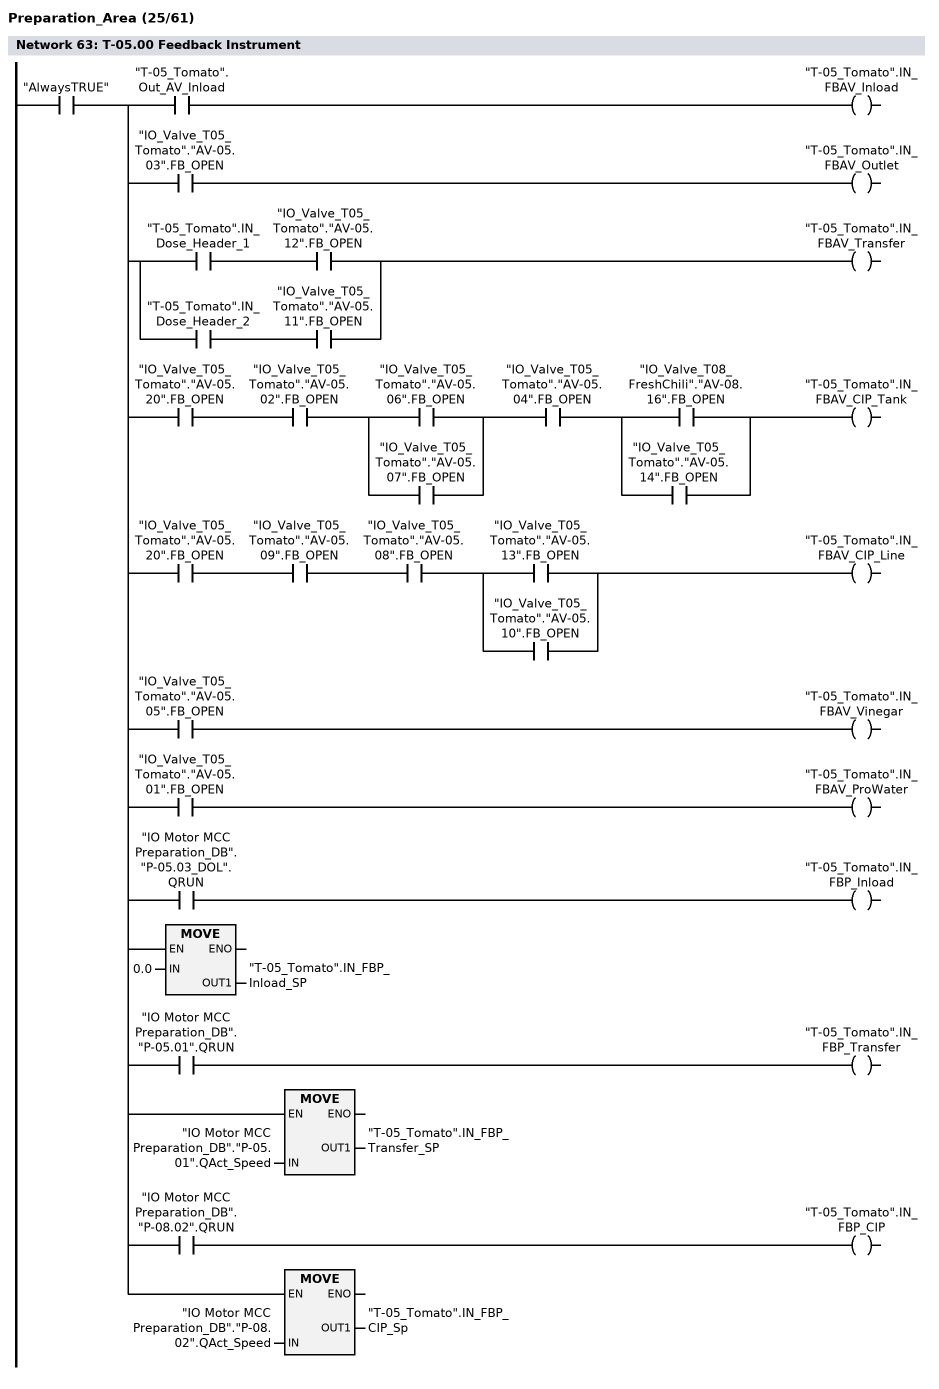
   RUNG wire#powerrail
      Contact( "AlwaysTRUE" )
      wire#w1
      Contact( "T-05_Tomato".Out_AV_Inload )
      Coil( "T-05_Tomato".IN_FBAV_Inload )
   END_RUNG
   RUNG wire#w1
      Contact( "IO_Valve_T05_Tomato"."AV-05.03".FB_OPEN )
      Coil( "T-05_Tomato".IN_FBAV_Outlet )
   END_RUNG
   RUNG wire#w1
      Contact( "T-05_Tomato".IN_Dose_Header_1 )
      Contact( "IO_Valve_T05_Tomato"."AV-05.12".FB_OPEN )
      wire#w2
      Coil( "T-05_Tomato".IN_FBAV_Transfer )
   END_RUNG
   RUNG wire#w1
      Contact( "T-05_Tomato".IN_Dose_Header_2 )
      Contact( "IO_Valve_T05_Tomato"."AV-05.11".FB_OPEN )
   END_RUNG wire#w2
   RUNG wire#w1
      Contact( "IO_Valve_T05_Tomato"."AV-05.20".FB_OPEN )
      Contact( "IO_Valve_T05_Tomato"."AV-05.02".FB_OPEN )
      wire#w3
      Contact( "IO_Valve_T05_Tomato"."AV-05.06".FB_OPEN )
      wire#w4
      Contact( "IO_Valve_T05_Tomato"."AV-05.04".FB_OPEN )
      wire#w5
      Contact( "IO_Valve_T08_FreshChili"."AV-08.16".FB_OPEN )
      wire#w6
      Coil( "T-05_Tomato".IN_FBAV_CIP_Tank )
   END_RUNG
   RUNG wire#w3
      Contact( "IO_Valve_T05_Tomato"."AV-05.07".FB_OPEN )
   END_RUNG wire#w4
   RUNG wire#w5
      Contact( "IO_Valve_T05_Tomato"."AV-05.14".FB_OPEN )
   END_RUNG wire#w6
   RUNG wire#w1
      Contact( "IO_Valve_T05_Tomato"."AV-05.20".FB_OPEN )
      Contact( "IO_Valve_T05_Tomato"."AV-05.09".FB_OPEN )
      Contact( "IO_Valve_T05_Tomato"."AV-05.08".FB_OPEN )
      wire#w7
      Contact( "IO_Valve_T05_Tomato"."AV-05.13".FB_OPEN )
      wire#w8
      Coil( "T-05_Tomato".IN_FBAV_CIP_Line )
   END_RUNG
   RUNG wire#w7
      Contact( "IO_Valve_T05_Tomato"."AV-05.10".FB_OPEN )
   END_RUNG wire#w8
   RUNG wire#w1
      Contact( "IO_Valve_T05_Tomato"."AV-05.05".FB_OPEN )
      Coil( "T-05_Tomato".IN_FBAV_Vinegar )
   END_RUNG
   RUNG wire#w1
      Contact( "IO_Valve_T05_Tomato"."AV-05.01".FB_OPEN )
      Coil( "T-05_Tomato".IN_FBAV_ProWater )
   END_RUNG
   RUNG wire#w1
      Contact( "IO Motor MCC Preparation_DB"."P-05.03_DOL".QRUN )
      Coil( "T-05_Tomato".IN_FBP_Inload )
   END_RUNG
   RUNG wire#w1
      Move(in := 0.0, out1 => "T-05_Tomato".IN_FBP_Inload_SP)
   END_RUNG
   RUNG wire#w1
      Contact( "IO Motor MCC Preparation_DB"."P-05.01".QRUN )
      Coil( "T-05_Tomato".IN_FBP_Transfer )
   END_RUNG
   RUNG wire#w1
      Move(in := "IO Motor MCC Preparation_DB"."P-05.01".QAct_Speed, out1 => "T-05_Tomato".IN_FBP_Transfer_SP)
   END_RUNG
   RUNG wire#w1
      Contact( "IO Motor MCC Preparation_DB"."P-08.02".QRUN )
      Coil( "T-05_Tomato".IN_FBP_CIP )
   END_RUNG
   RUNG wire#w1
      Move(in := "IO Motor MCC Preparation_DB"."P-08.02".QAct_Speed, out1 => "T-05_Tomato".IN_FBP_CIP_Sp)
   END_RUNG
   // the same network as SCL:
   "T-05_Tomato".IN_FBAV_Inload := "AlwaysTRUE" AND "T-05_Tomato".Out_AV_Inload;
   "T-05_Tomato".IN_FBAV_Outlet := "AlwaysTRUE" AND "IO_Valve_T05_Tomato"."AV-05.03".FB_OPEN;
   "T-05_Tomato".IN_FBAV_Transfer := "AlwaysTRUE" AND (("T-05_Tomato".IN_Dose_Header_1 AND "IO_Valve_T05_Tomato"."AV-05.12".FB_OPEN) OR ("T-05_Tomato".IN_Dose_Header_2 AND "IO_Valve_T05_Tomato"."AV-05.11".FB_OPEN));
   "T-05_Tomato".IN_FBAV_CIP_Tank := "AlwaysTRUE" AND "IO_Valve_T05_Tomato"."AV-05.20".FB_OPEN AND "IO_Valve_T05_Tomato"."AV-05.02".FB_OPEN AND ("IO_Valve_T05_Tomato"."AV-05.06".FB_OPEN OR "IO_Valve_T05_Tomato"."AV-05.07".FB_OPEN) AND "IO_Valve_T05_Tomato"."AV-05.04".FB_OPEN AND ("IO_Valve_T08_FreshChili"."AV-08.16".FB_OPEN OR "IO_Valve_T05_Tomato"."AV-05.14".FB_OPEN);
   "T-05_Tomato".IN_FBAV_CIP_Line := "AlwaysTRUE" AND "IO_Valve_T05_Tomato"."AV-05.20".FB_OPEN AND "IO_Valve_T05_Tomato"."AV-05.09".FB_OPEN AND "IO_Valve_T05_Tomato"."AV-05.08".FB_OPEN AND ("IO_Valve_T05_Tomato"."AV-05.13".FB_OPEN OR "IO_Valve_T05_Tomato"."AV-05.10".FB_OPEN);
   "T-05_Tomato".IN_FBAV_Vinegar := "AlwaysTRUE" AND "IO_Valve_T05_Tomato"."AV-05.05".FB_OPEN;
   "T-05_Tomato".IN_FBAV_ProWater := "AlwaysTRUE" AND "IO_Valve_T05_Tomato"."AV-05.01".FB_OPEN;
   "T-05_Tomato".IN_FBP_Inload := "AlwaysTRUE" AND "IO Motor MCC Preparation_DB"."P-05.03_DOL".QRUN;
   IF "AlwaysTRUE" THEN "T-05_Tomato".IN_FBP_Inload_SP := 0.0; END_IF;
   "T-05_Tomato".IN_FBP_Transfer := "AlwaysTRUE" AND "IO Motor MCC Preparation_DB"."P-05.01".QRUN;
   IF "AlwaysTRUE" THEN
       "T-05_Tomato".IN_FBP_Transfer_SP := "IO Motor MCC Preparation_DB"."P-05.01".QAct_Speed;
   END_IF;
   "T-05_Tomato".IN_FBP_CIP := "AlwaysTRUE" AND "IO Motor MCC Preparation_DB"."P-08.02".QRUN;
   IF "AlwaysTRUE" THEN
       "T-05_Tomato".IN_FBP_CIP_Sp := "IO Motor MCC Preparation_DB"."P-08.02".QAct_Speed;
   END_IF;
END_REGION

REGION Network 64: T-05.00 Comm to Blend
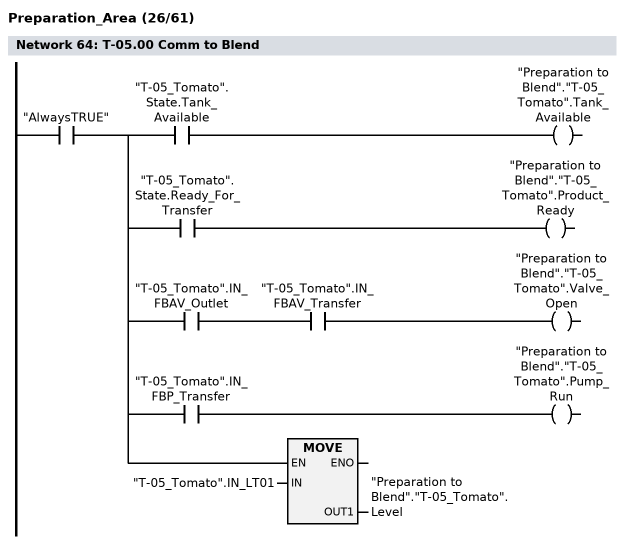
   RUNG wire#powerrail
      Contact( "AlwaysTRUE" )
      wire#w1
      Contact( "T-05_Tomato".State.Tank_Available )
      Coil( "Preparation to Blend"."T-05_Tomato".Tank_Available )
   END_RUNG
   RUNG wire#w1
      Contact( "T-05_Tomato".State.Ready_For_Transfer )
      Coil( "Preparation to Blend"."T-05_Tomato".Product_Ready )
   END_RUNG
   RUNG wire#w1
      Contact( "T-05_Tomato".IN_FBAV_Outlet )
      Contact( "T-05_Tomato".IN_FBAV_Transfer )
      Coil( "Preparation to Blend"."T-05_Tomato".Valve_Open )
   END_RUNG
   RUNG wire#w1
      Contact( "T-05_Tomato".IN_FBP_Transfer )
      Coil( "Preparation to Blend"."T-05_Tomato".Pump_Run )
   END_RUNG
   RUNG wire#w1
      Move(in := "T-05_Tomato".IN_LT01, out1 => "Preparation to Blend"."T-05_Tomato".Level)
   END_RUNG
   // the same network as SCL:
   "Preparation to Blend"."T-05_Tomato".Tank_Available := "AlwaysTRUE" AND "T-05_Tomato".State.Tank_Available;
   "Preparation to Blend"."T-05_Tomato".Product_Ready := "AlwaysTRUE" AND "T-05_Tomato".State.Ready_For_Transfer;
   "Preparation to Blend"."T-05_Tomato".Valve_Open := "AlwaysTRUE" AND "T-05_Tomato".IN_FBAV_Outlet AND "T-05_Tomato".IN_FBAV_Transfer;
   "Preparation to Blend"."T-05_Tomato".Pump_Run := "AlwaysTRUE" AND "T-05_Tomato".IN_FBP_Transfer;
   IF "AlwaysTRUE" THEN "Preparation to Blend"."T-05_Tomato".Level := "T-05_Tomato".IN_LT01; END_IF;
END_REGION

NETWORK
TITLE = T-06.00 DOSE ON OFF
      O     "Blend to Preparation"."T-20".Raw_Material.ChiliFresh_1.DoseRun;
      O     "Blend to Preparation"."T-21".Raw_Material.ChiliFresh_1.DoseRun;
      O     "Blend to Preparation"."T-30".Raw_Material.ChiliFresh_1.DoseRun;
      O     "Blend to Preparation"."T-31".Raw_Material.ChiliFresh_1.DoseRun;
      O     "Blend to Preparation"."T-40".Raw_Material.ChiliFresh_1.DoseRun;
      O     "Blend to Preparation"."T-41".Raw_Material.ChiliFresh_1.DoseRun;
      =     "T-06_ChiliFresh_1".IN_Dose_Run;

NETWORK
TITLE = T-06.00 DOSE PAUSE
      O     "Blend to Preparation"."T-20".Raw_Material.ChiliFresh_1.DoseHeld;
      O     "Blend to Preparation"."T-21".Raw_Material.ChiliFresh_1.DoseHeld;
      O     "Blend to Preparation"."T-30".Raw_Material.ChiliFresh_1.DoseHeld;
      O     "Blend to Preparation"."T-31".Raw_Material.ChiliFresh_1.DoseHeld;
      O     "Blend to Preparation"."T-40".Raw_Material.ChiliFresh_1.DoseHeld;
      O     "Blend to Preparation"."T-41".Raw_Material.ChiliFresh_1.DoseHeld;
      =     "T-06_ChiliFresh_1".IN_Dose_Held;

NETWORK
TITLE = T-06.00 DOSE VALVE CMD
      O(;
      A     "Blend to Preparation"."T-20".Raw_Material.ChiliFresh_1.DoseRun;
      A     "Blend to Preparation"."T-20".Raw_Material.ChiliFresh_1.ValveCMD;
      );
      O(;
      A     "Blend to Preparation"."T-21".Raw_Material.ChiliFresh_1.DoseRun;
      A     "Blend to Preparation"."T-21".Raw_Material.ChiliFresh_1.ValveCMD;
      );
      O(;
      A     "Blend to Preparation"."T-30".Raw_Material.ChiliFresh_1.DoseRun;
      A     "Blend to Preparation"."T-30".Raw_Material.ChiliFresh_1.ValveCMD;
      );
      O(;
      A     "Blend to Preparation"."T-31".Raw_Material.ChiliFresh_1.DoseRun;
      A     "Blend to Preparation"."T-31".Raw_Material.ChiliFresh_1.ValveCMD;
      );
      O(;
      A     "Blend to Preparation"."T-40".Raw_Material.ChiliFresh_1.DoseRun;
      A     "Blend to Preparation"."T-40".Raw_Material.ChiliFresh_1.ValveCMD;
      );
      O(;
      A     "Blend to Preparation"."T-41".Raw_Material.ChiliFresh_1.DoseRun;
      A     "Blend to Preparation"."T-41".Raw_Material.ChiliFresh_1.ValveCMD;
      );
      =     "T-06_ChiliFresh_1".IN_Dose_Valve_Cmd;



NETWORK
TITLE = T-06.00 DOSE Pump CMD
      O(;
      A     "Blend to Preparation"."T-20".Raw_Material.ChiliFresh_1.DoseRun;
      A     "Blend to Preparation"."T-20".Raw_Material.ChiliFresh_1.PumpCMD;
      );
      O(;
      A     "Blend to Preparation"."T-21".Raw_Material.ChiliFresh_1.DoseRun;
      A     "Blend to Preparation"."T-21".Raw_Material.ChiliFresh_1.PumpCMD;
      );
      O(;
      A     "Blend to Preparation"."T-30".Raw_Material.ChiliFresh_1.DoseRun;
      A     "Blend to Preparation"."T-30".Raw_Material.ChiliFresh_1.PumpCMD;
      );
      O(;
      A     "Blend to Preparation"."T-31".Raw_Material.ChiliFresh_1.DoseRun;
      A     "Blend to Preparation"."T-31".Raw_Material.ChiliFresh_1.PumpCMD;
      );
      O(;
      A     "Blend to Preparation"."T-40".Raw_Material.ChiliFresh_1.DoseRun;
      A     "Blend to Preparation"."T-40".Raw_Material.ChiliFresh_1.PumpCMD;
      );
      O(;
      A     "Blend to Preparation"."T-41".Raw_Material.ChiliFresh_1.DoseRun;
      A     "Blend to Preparation"."T-41".Raw_Material.ChiliFresh_1.PumpCMD;
      );
      =     "T-06_ChiliFresh_1".IN_Dose_Pump_Cmd;



NETWORK
TITLE = T-06.00 DOSE PUMP SPEED
// Checking
      O     "Blend to Preparation"."T-20".Raw_Material.ChiliFresh_1.DoseRun;
      JC    SP_06_FROM_20;
      O     "Blend to Preparation"."T-21".Raw_Material.ChiliFresh_1.DoseRun;
      JC    SP_06_FROM_21;
      O     "Blend to Preparation"."T-30".Raw_Material.ChiliFresh_1.DoseRun;
      JC    SP_06_FROM_30;
      O     "Blend to Preparation"."T-31".Raw_Material.ChiliFresh_1.DoseRun;
      JC    SP_06_FROM_31;
      O     "Blend to Preparation"."T-40".Raw_Material.ChiliFresh_1.DoseRun;
      JC    SP_06_FROM_40;
      O     "Blend to Preparation"."T-41".Raw_Material.ChiliFresh_1.DoseRun;
      JC    SP_06_FROM_41;
//Jump to end if Blend not Dosing
      JC    SP_06_SELF;
//Load Set Point
SP_06_FROM_20:L     "Blend to Preparation".Recipe."T-20".ChiliFresh_1.SP_PumpSpeed;
      T     "T-06_ChiliFresh_1".IN_Dose_Pump_Sp;
      JC    SP_06_SELF;
SP_06_FROM_21:L     "Blend to Preparation".Recipe."T-21".ChiliFresh_1.SP_PumpSpeed;
      T     "T-06_ChiliFresh_1".IN_Dose_Pump_Sp;
      JC    SP_06_SELF;
SP_06_FROM_30:L     "Blend to Preparation".Recipe."T-30".ChiliFresh_1.SP_PumpSpeed;
      T     "T-06_ChiliFresh_1".IN_Dose_Pump_Sp;
      JC    SP_06_SELF;
SP_06_FROM_31:L     "Blend to Preparation".Recipe."T-31".ChiliFresh_1.SP_PumpSpeed;
      T     "T-06_ChiliFresh_1".IN_Dose_Pump_Sp;
      JC    SP_06_SELF;
SP_06_FROM_40:L     "Blend to Preparation".Recipe."T-40".ChiliFresh_1.SP_PumpSpeed;
      T     "T-06_ChiliFresh_1".IN_Dose_Pump_Sp;
      JC    SP_06_SELF;
SP_06_FROM_41:L     "Blend to Preparation".Recipe."T-41".ChiliFresh_1.SP_PumpSpeed;
      T     "T-06_ChiliFresh_1".IN_Dose_Pump_Sp;
      JC    SP_06_SELF;
// END
SP_06_SELF:L     "T-06_ChiliFresh_1".IN_Dose_Pump_Sp;
      T     "T-06_ChiliFresh_1".IN_Dose_Pump_Sp;


NETWORK
TITLE = T-06.00 Header Req
// HEADER 1 Req
      O     "Blend to Preparation"."T-20".Raw_Material.ChiliFresh_1.Header1_Req;
      O     "Blend to Preparation"."T-21".Raw_Material.ChiliFresh_1.Header1_Req;
      O     "Blend to Preparation"."T-30".Raw_Material.ChiliFresh_1.Header1_Req;
      O     "Blend to Preparation"."T-31".Raw_Material.ChiliFresh_1.Header1_Req;
      O     "Blend to Preparation"."T-40".Raw_Material.ChiliFresh_1.Header1_Req;
      O     "Blend to Preparation"."T-41".Raw_Material.ChiliFresh_1.Header1_Req;
      =     "T-06_ChiliFresh_1".IN_Dose_Header_1;

// HEADER 2 Req
      O     "Blend to Preparation"."T-20".Raw_Material.ChiliFresh_1.Header2_Req;
      O     "Blend to Preparation"."T-21".Raw_Material.ChiliFresh_1.Header2_Req;
      O     "Blend to Preparation"."T-30".Raw_Material.ChiliFresh_1.Header2_Req;
      O     "Blend to Preparation"."T-31".Raw_Material.ChiliFresh_1.Header2_Req;
      O     "Blend to Preparation"."T-40".Raw_Material.ChiliFresh_1.Header2_Req;
      O     "Blend to Preparation"."T-41".Raw_Material.ChiliFresh_1.Header2_Req;
      =     "T-06_ChiliFresh_1".IN_Dose_Header_2;


REGION Network 73: T-06.00 LineTransferOK
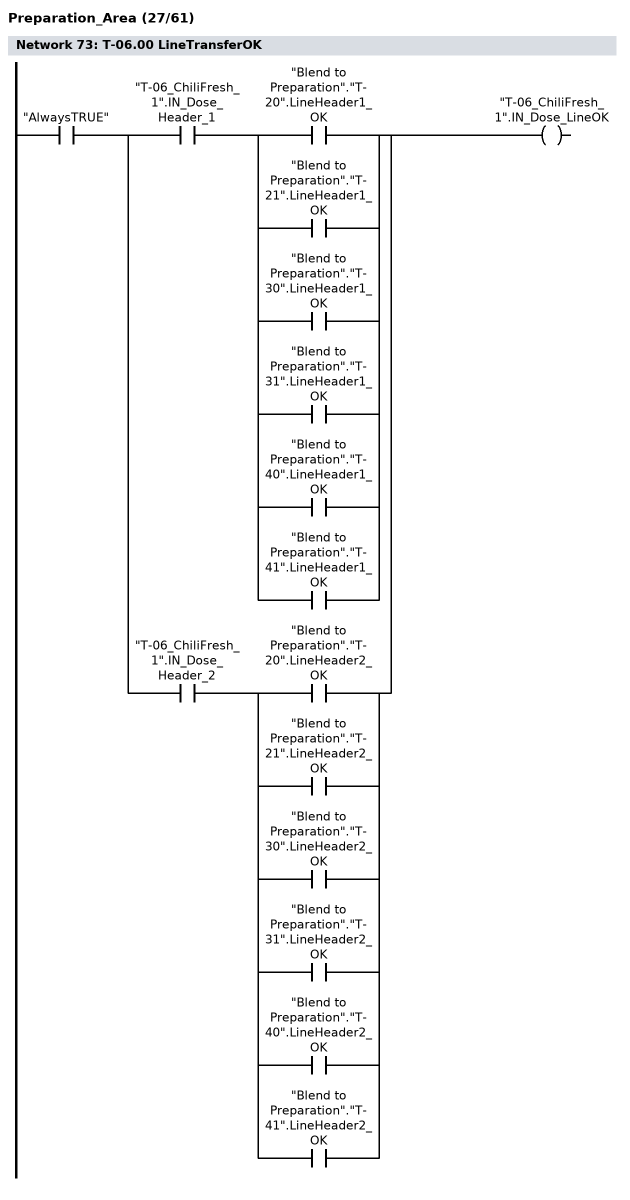
   RUNG wire#powerrail
      Contact( "AlwaysTRUE" )
      wire#w1
      Contact( "T-06_ChiliFresh_1".IN_Dose_Header_1 )
      wire#w2
      Contact( "Blend to Preparation"."T-20".LineHeader1_OK )
      wire#w3
      Coil( "T-06_ChiliFresh_1".IN_Dose_LineOK )
   END_RUNG
   RUNG wire#w2
      Contact( "Blend to Preparation"."T-21".LineHeader1_OK )
   END_RUNG wire#w3
   RUNG wire#w2
      Contact( "Blend to Preparation"."T-30".LineHeader1_OK )
   END_RUNG wire#w3
   RUNG wire#w2
      Contact( "Blend to Preparation"."T-31".LineHeader1_OK )
   END_RUNG wire#w3
   RUNG wire#w2
      Contact( "Blend to Preparation"."T-40".LineHeader1_OK )
   END_RUNG wire#w3
   RUNG wire#w2
      Contact( "Blend to Preparation"."T-41".LineHeader1_OK )
   END_RUNG wire#w3
   RUNG wire#w1
      Contact( "T-06_ChiliFresh_1".IN_Dose_Header_2 )
      wire#w4
      Contact( "Blend to Preparation"."T-20".LineHeader2_OK )
   END_RUNG wire#w3
   RUNG wire#w4
      Contact( "Blend to Preparation"."T-21".LineHeader2_OK )
   END_RUNG wire#w3
   RUNG wire#w4
      Contact( "Blend to Preparation"."T-30".LineHeader2_OK )
   END_RUNG wire#w3
   RUNG wire#w4
      Contact( "Blend to Preparation"."T-31".LineHeader2_OK )
   END_RUNG wire#w3
   RUNG wire#w4
      Contact( "Blend to Preparation"."T-40".LineHeader2_OK )
   END_RUNG wire#w3
   RUNG wire#w4
      Contact( "Blend to Preparation"."T-41".LineHeader2_OK )
   END_RUNG wire#w3
   // the same network as SCL:
   "T-06_ChiliFresh_1".IN_Dose_LineOK := "AlwaysTRUE" AND (("T-06_ChiliFresh_1".IN_Dose_Header_1 AND ("Blend to Preparation"."T-20".LineHeader1_OK OR "Blend to Preparation"."T-21".LineHeader1_OK OR "Blend to Preparation"."T-30".LineHeader1_OK OR "Blend to Preparation"."T-31".LineHeader1_OK OR "Blend to Preparation"."T-40".LineHeader1_OK OR "Blend to Preparation"."T-41".LineHeader1_OK)) OR ("T-06_ChiliFresh_1".IN_Dose_Header_2 AND ("Blend to Preparation"."T-20".LineHeader2_OK OR "Blend to Preparation"."T-21".LineHeader2_OK OR "Blend to Preparation"."T-30".LineHeader2_OK OR "Blend to Preparation"."T-31".LineHeader2_OK OR "Blend to Preparation"."T-40".LineHeader2_OK OR "Blend to Preparation"."T-41".LineHeader2_OK)));
END_REGION

REGION Network 74: T-06____Chili Fresh 1
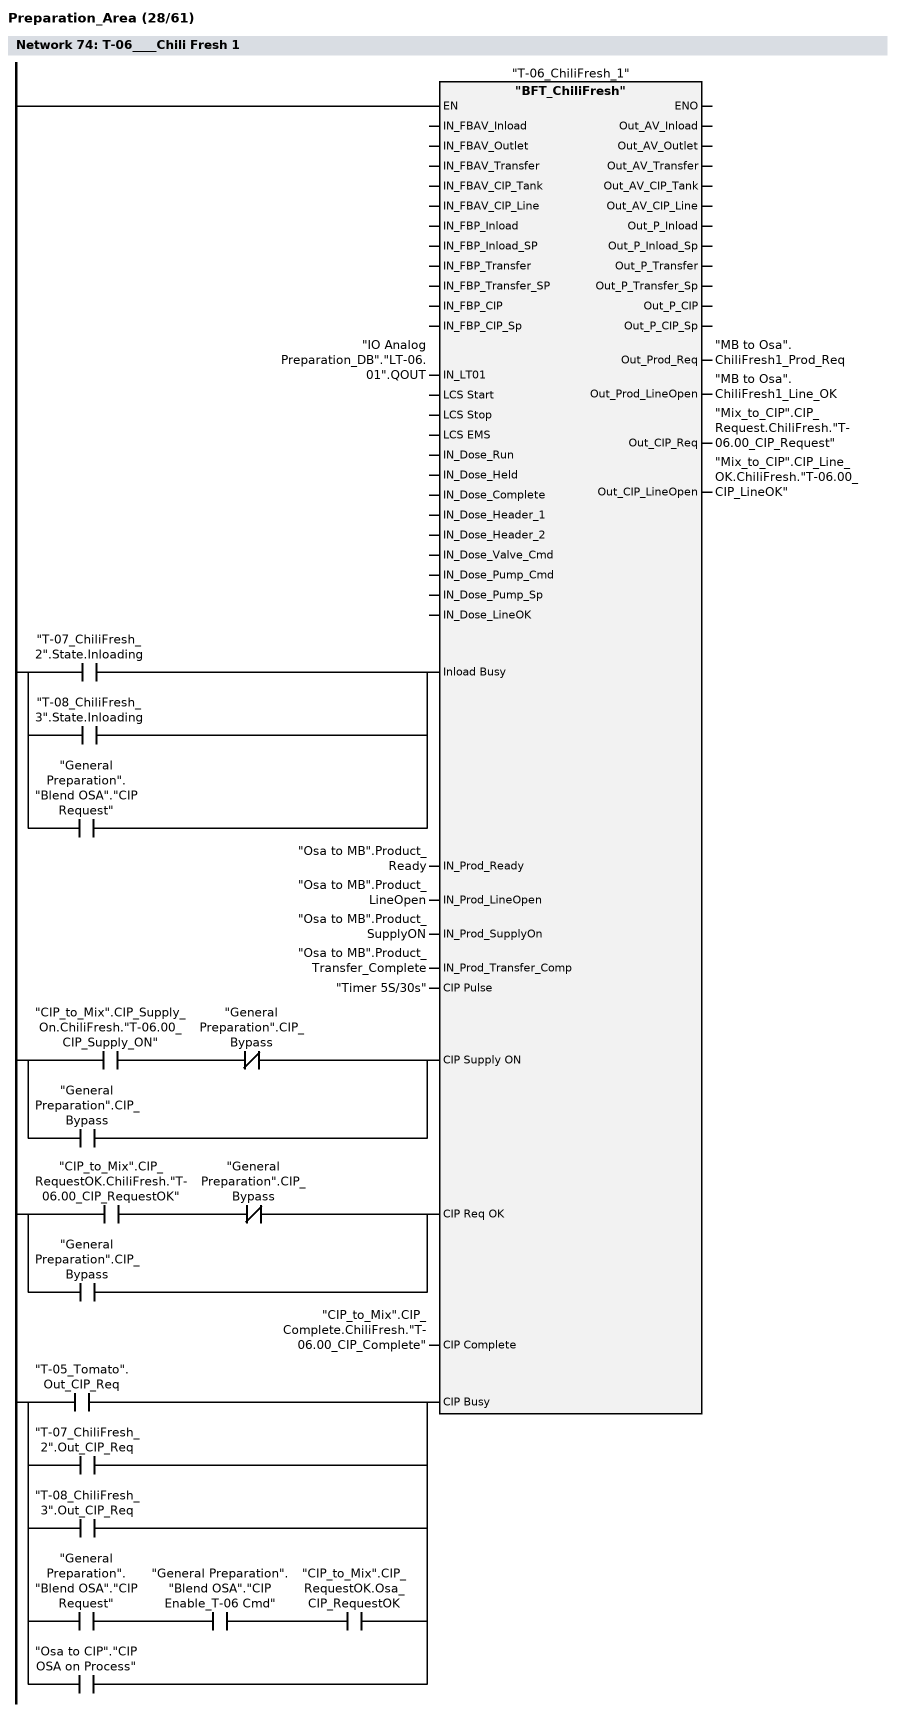
   RUNG wire#powerrail
      "T-06_ChiliFresh_1"("Inload Busy" := wire#w1, "CIP Supply ON" := wire#w2, "CIP Req OK" := wire#w3, "CIP Busy" := wire#w4, IN_FBAV_Inload :=, IN_FBAV_Outlet :=, IN_FBAV_Transfer :=, IN_FBAV_CIP_Tank :=, IN_FBAV_CIP_Line :=, IN_FBP_Inload :=, IN_FBP_Inload_SP :=, IN_FBP_Transfer :=, IN_FBP_Transfer_SP :=, IN_FBP_CIP :=, IN_FBP_CIP_Sp :=, IN_LT01 := "IO Analog Preparation_DB"."LT-06.01".QOUT, "LCS Start" :=, "LCS Stop" :=, "LCS EMS" :=, IN_Dose_Run :=, IN_Dose_Held :=, IN_Dose_Complete :=, IN_Dose_Header_1 :=, IN_Dose_Header_2 :=, IN_Dose_Valve_Cmd :=, IN_Dose_Pump_Cmd :=, IN_Dose_Pump_Sp :=, IN_Dose_LineOK :=, IN_Prod_Ready := "Osa to MB".Product_Ready, IN_Prod_LineOpen := "Osa to MB".Product_LineOpen, IN_Prod_SupplyOn := "Osa to MB".Product_SupplyON, IN_Prod_Transfer_Comp := "Osa to MB".Product_Transfer_Complete, "CIP Pulse" := "Timer 5S/30s", "CIP Complete" := "CIP_to_Mix".CIP_Complete.ChiliFresh."T-06.00_CIP_Complete", Out_AV_Inload =>, Out_AV_Outlet =>, Out_AV_Transfer =>, Out_AV_CIP_Tank =>, Out_AV_CIP_Line =>, Out_P_Inload =>, Out_P_Inload_Sp =>, Out_P_Transfer =>, Out_P_Transfer_Sp =>, Out_P_CIP =>, Out_P_CIP_Sp =>, Out_Prod_Req => "MB to Osa".ChiliFresh1_Prod_Req, Out_Prod_LineOpen => "MB to Osa".ChiliFresh1_Line_OK, Out_CIP_Req => "Mix_to_CIP".CIP_Request.ChiliFresh."T-06.00_CIP_Request", Out_CIP_LineOpen => "Mix_to_CIP".CIP_Line_OK.ChiliFresh."T-06.00_CIP_LineOK")
   END_RUNG
   RUNG wire#powerrail
      Contact( "T-07_ChiliFresh_2".State.Inloading )
   END_RUNG wire#w1
   RUNG wire#powerrail
      Contact( "T-08_ChiliFresh_3".State.Inloading )
   END_RUNG wire#w1
   RUNG wire#powerrail
      Contact( "General Preparation"."Blend OSA"."CIP Request" )
   END_RUNG wire#w1
   RUNG wire#powerrail
      Contact( "CIP_to_Mix".CIP_Supply_On.ChiliFresh."T-06.00_CIP_Supply_ON" )
      I_Contact( "General Preparation".CIP_Bypass )
   END_RUNG wire#w2
   RUNG wire#powerrail
      Contact( "General Preparation".CIP_Bypass )
   END_RUNG wire#w2
   RUNG wire#powerrail
      Contact( "CIP_to_Mix".CIP_RequestOK.ChiliFresh."T-06.00_CIP_RequestOK" )
      I_Contact( "General Preparation".CIP_Bypass )
   END_RUNG wire#w3
   RUNG wire#powerrail
      Contact( "General Preparation".CIP_Bypass )
   END_RUNG wire#w3
   RUNG wire#powerrail
      Contact( "T-05_Tomato".Out_CIP_Req )
   END_RUNG wire#w4
   RUNG wire#powerrail
      Contact( "T-07_ChiliFresh_2".Out_CIP_Req )
   END_RUNG wire#w4
   RUNG wire#powerrail
      Contact( "T-08_ChiliFresh_3".Out_CIP_Req )
   END_RUNG wire#w4
   RUNG wire#powerrail
      Contact( "General Preparation"."Blend OSA"."CIP Request" )
      Contact( "General Preparation"."Blend OSA"."CIP Enable_T-06 Cmd" )
      Contact( "CIP_to_Mix".CIP_RequestOK.Osa_CIP_RequestOK )
   END_RUNG wire#w4
   RUNG wire#powerrail
      Contact( "Osa to CIP"."CIP OSA on Process" )
   END_RUNG wire#w4
   // the same network as SCL:
   "T-06_ChiliFresh_1"(IN_LT01 := "IO Analog Preparation_DB"."LT-06.01".QOUT,   // "BFT_ChiliFresh"
                       "Inload Busy" := "T-07_ChiliFresh_2".State.Inloading OR "T-08_ChiliFresh_3".State.Inloading OR "General Preparation"."Blend OSA"."CIP Request",
                       IN_Prod_Ready := "Osa to MB".Product_Ready,
                       IN_Prod_LineOpen := "Osa to MB".Product_LineOpen,
                       IN_Prod_SupplyOn := "Osa to MB".Product_SupplyON,
                       IN_Prod_Transfer_Comp := "Osa to MB".Product_Transfer_Complete,
                       "CIP Pulse" := "Timer 5S/30s",
                       "CIP Supply ON" := ("CIP_to_Mix".CIP_Supply_On.ChiliFresh."T-06.00_CIP_Supply_ON" AND NOT "General Preparation".CIP_Bypass) OR "General Preparation".CIP_Bypass,
                       "CIP Req OK" := ("CIP_to_Mix".CIP_RequestOK.ChiliFresh."T-06.00_CIP_RequestOK" AND NOT "General Preparation".CIP_Bypass) OR "General Preparation".CIP_Bypass,
                       "CIP Complete" := "CIP_to_Mix".CIP_Complete.ChiliFresh."T-06.00_CIP_Complete",
                       "CIP Busy" := "T-05_Tomato".Out_CIP_Req OR "T-07_ChiliFresh_2".Out_CIP_Req OR "T-08_ChiliFresh_3".Out_CIP_Req OR ("General Preparation"."Blend OSA"."CIP Request" AND "General Preparation"."Blend OSA"."CIP Enable_T-06 Cmd" AND "CIP_to_Mix".CIP_RequestOK.Osa_CIP_RequestOK) OR "Osa to CIP"."CIP OSA on Process",
                       Out_Prod_Req => "MB to Osa".ChiliFresh1_Prod_Req,
                       Out_Prod_LineOpen => "MB to Osa".ChiliFresh1_Line_OK,
                       Out_CIP_Req => "Mix_to_CIP".CIP_Request.ChiliFresh."T-06.00_CIP_Request",
                       Out_CIP_LineOpen => "Mix_to_CIP".CIP_Line_OK.ChiliFresh."T-06.00_CIP_LineOK");
END_REGION

REGION Network 75: T-06.00 Valve Cmd
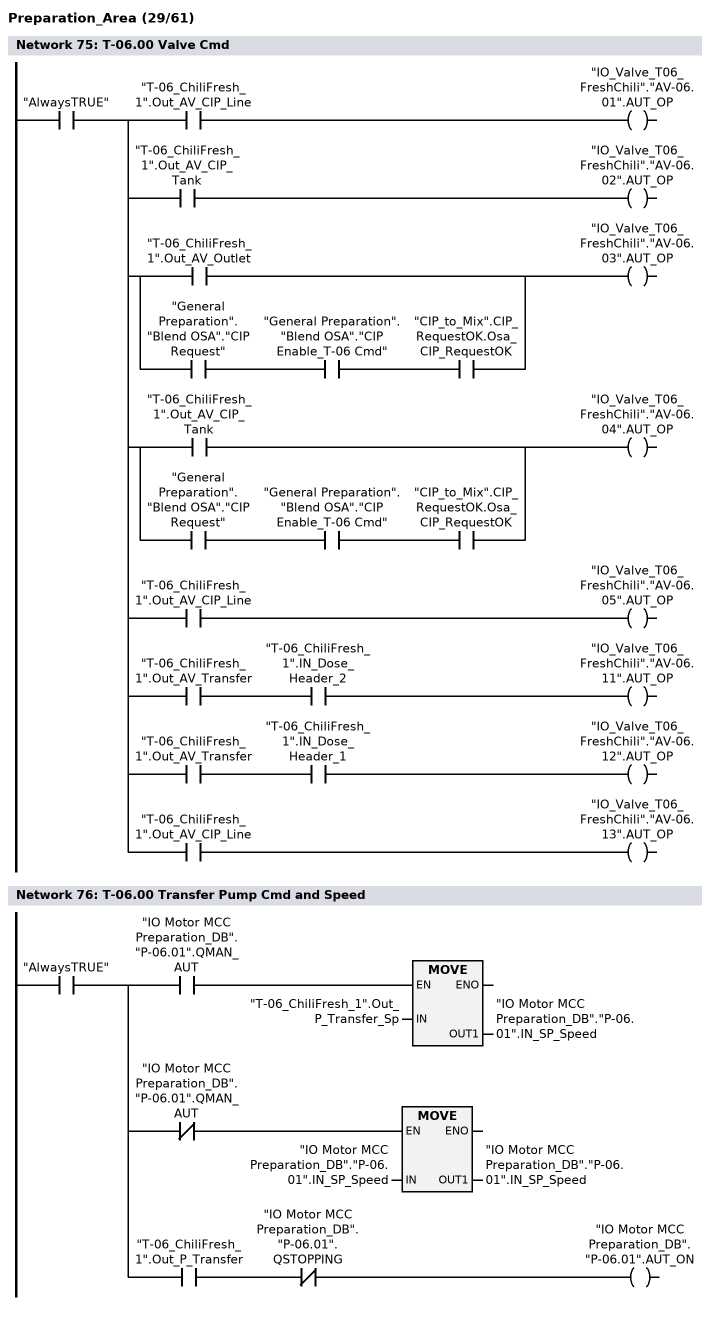
   RUNG wire#powerrail
      Contact( "AlwaysTRUE" )
      wire#w1
      Contact( "T-06_ChiliFresh_1".Out_AV_CIP_Line )
      Coil( "IO_Valve_T06_FreshChili"."AV-06.01".AUT_OP )
   END_RUNG
   RUNG wire#w1
      Contact( "T-06_ChiliFresh_1".Out_AV_CIP_Tank )
      Coil( "IO_Valve_T06_FreshChili"."AV-06.02".AUT_OP )
   END_RUNG
   RUNG wire#w1
      Contact( "T-06_ChiliFresh_1".Out_AV_Outlet )
      wire#w2
      Coil( "IO_Valve_T06_FreshChili"."AV-06.03".AUT_OP )
   END_RUNG
   RUNG wire#w1
      Contact( "General Preparation"."Blend OSA"."CIP Request" )
      Contact( "General Preparation"."Blend OSA"."CIP Enable_T-06 Cmd" )
      Contact( "CIP_to_Mix".CIP_RequestOK.Osa_CIP_RequestOK )
   END_RUNG wire#w2
   RUNG wire#w1
      Contact( "T-06_ChiliFresh_1".Out_AV_CIP_Tank )
      wire#w3
      Coil( "IO_Valve_T06_FreshChili"."AV-06.04".AUT_OP )
   END_RUNG
   RUNG wire#w1
      Contact( "General Preparation"."Blend OSA"."CIP Request" )
      Contact( "General Preparation"."Blend OSA"."CIP Enable_T-06 Cmd" )
      Contact( "CIP_to_Mix".CIP_RequestOK.Osa_CIP_RequestOK )
   END_RUNG wire#w3
   RUNG wire#w1
      Contact( "T-06_ChiliFresh_1".Out_AV_CIP_Line )
      Coil( "IO_Valve_T06_FreshChili"."AV-06.05".AUT_OP )
   END_RUNG
   RUNG wire#w1
      Contact( "T-06_ChiliFresh_1".Out_AV_Transfer )
      Contact( "T-06_ChiliFresh_1".IN_Dose_Header_2 )
      Coil( "IO_Valve_T06_FreshChili"."AV-06.11".AUT_OP )
   END_RUNG
   RUNG wire#w1
      Contact( "T-06_ChiliFresh_1".Out_AV_Transfer )
      Contact( "T-06_ChiliFresh_1".IN_Dose_Header_1 )
      Coil( "IO_Valve_T06_FreshChili"."AV-06.12".AUT_OP )
   END_RUNG
   RUNG wire#w1
      Contact( "T-06_ChiliFresh_1".Out_AV_CIP_Line )
      Coil( "IO_Valve_T06_FreshChili"."AV-06.13".AUT_OP )
   END_RUNG
   // the same network as SCL:
   "IO_Valve_T06_FreshChili"."AV-06.01".AUT_OP := "AlwaysTRUE" AND "T-06_ChiliFresh_1".Out_AV_CIP_Line;
   "IO_Valve_T06_FreshChili"."AV-06.02".AUT_OP := "AlwaysTRUE" AND "T-06_ChiliFresh_1".Out_AV_CIP_Tank;
   "IO_Valve_T06_FreshChili"."AV-06.03".AUT_OP := "AlwaysTRUE" AND ("T-06_ChiliFresh_1".Out_AV_Outlet OR ("General Preparation"."Blend OSA"."CIP Request" AND "General Preparation"."Blend OSA"."CIP Enable_T-06 Cmd" AND "CIP_to_Mix".CIP_RequestOK.Osa_CIP_RequestOK));
   "IO_Valve_T06_FreshChili"."AV-06.04".AUT_OP := "AlwaysTRUE" AND ("T-06_ChiliFresh_1".Out_AV_CIP_Tank OR ("General Preparation"."Blend OSA"."CIP Request" AND "General Preparation"."Blend OSA"."CIP Enable_T-06 Cmd" AND "CIP_to_Mix".CIP_RequestOK.Osa_CIP_RequestOK));
   "IO_Valve_T06_FreshChili"."AV-06.05".AUT_OP := "AlwaysTRUE" AND "T-06_ChiliFresh_1".Out_AV_CIP_Line;
   "IO_Valve_T06_FreshChili"."AV-06.11".AUT_OP := "AlwaysTRUE" AND "T-06_ChiliFresh_1".Out_AV_Transfer AND "T-06_ChiliFresh_1".IN_Dose_Header_2;
   "IO_Valve_T06_FreshChili"."AV-06.12".AUT_OP := "AlwaysTRUE" AND "T-06_ChiliFresh_1".Out_AV_Transfer AND "T-06_ChiliFresh_1".IN_Dose_Header_1;
   "IO_Valve_T06_FreshChili"."AV-06.13".AUT_OP := "AlwaysTRUE" AND "T-06_ChiliFresh_1".Out_AV_CIP_Line;
END_REGION

REGION Network 76: T-06.00 Transfer Pump Cmd and Speed
   RUNG wire#powerrail
      Contact( "AlwaysTRUE" )
      wire#w1
      Contact( "IO Motor MCC Preparation_DB"."P-06.01".QMAN_AUT )
      Move(in := "T-06_ChiliFresh_1".Out_P_Transfer_Sp, out1 => "IO Motor MCC Preparation_DB"."P-06.01".IN_SP_Speed)
   END_RUNG
   RUNG wire#w1
      I_Contact( "IO Motor MCC Preparation_DB"."P-06.01".QMAN_AUT )
      Move(in := "IO Motor MCC Preparation_DB"."P-06.01".IN_SP_Speed, out1 => "IO Motor MCC Preparation_DB"."P-06.01".IN_SP_Speed)
   END_RUNG
   RUNG wire#w1
      Contact( "T-06_ChiliFresh_1".Out_P_Transfer )
      I_Contact( "IO Motor MCC Preparation_DB"."P-06.01".QSTOPPING )
      Coil( "IO Motor MCC Preparation_DB"."P-06.01".AUT_ON )
   END_RUNG
   // the same network as SCL:
   IF "AlwaysTRUE" AND "IO Motor MCC Preparation_DB"."P-06.01".QMAN_AUT THEN
       "IO Motor MCC Preparation_DB"."P-06.01".IN_SP_Speed := "T-06_ChiliFresh_1".Out_P_Transfer_Sp;
   END_IF;
   IF "AlwaysTRUE" AND NOT "IO Motor MCC Preparation_DB"."P-06.01".QMAN_AUT THEN
       "IO Motor MCC Preparation_DB"."P-06.01".IN_SP_Speed := "IO Motor MCC Preparation_DB"."P-06.01".IN_SP_Speed;
   END_IF;
   "IO Motor MCC Preparation_DB"."P-06.01".AUT_ON := "AlwaysTRUE" AND "T-06_ChiliFresh_1".Out_P_Transfer AND NOT "IO Motor MCC Preparation_DB"."P-06.01".QSTOPPING;
END_REGION

REGION Network 77: T-06.00 Feedback Instrument
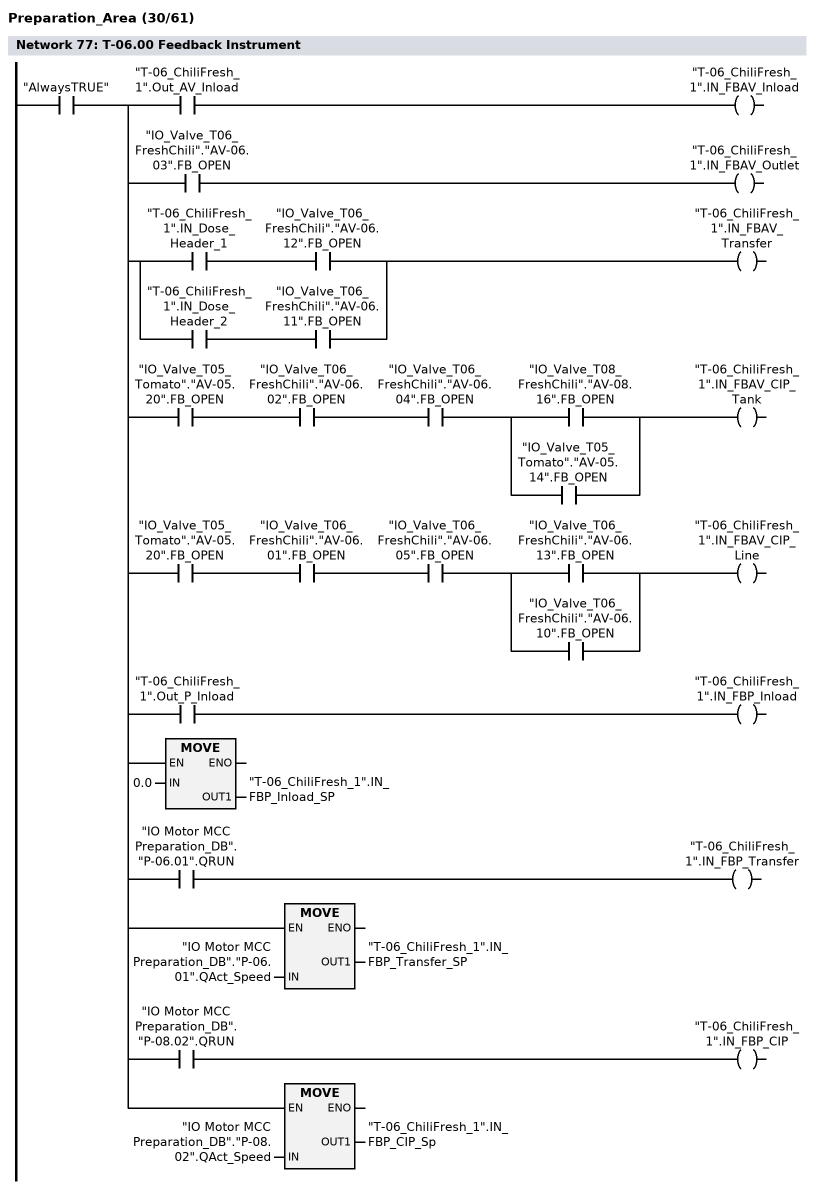
   RUNG wire#powerrail
      Contact( "AlwaysTRUE" )
      wire#w1
      Contact( "T-06_ChiliFresh_1".Out_AV_Inload )
      Coil( "T-06_ChiliFresh_1".IN_FBAV_Inload )
   END_RUNG
   RUNG wire#w1
      Contact( "IO_Valve_T06_FreshChili"."AV-06.03".FB_OPEN )
      Coil( "T-06_ChiliFresh_1".IN_FBAV_Outlet )
   END_RUNG
   RUNG wire#w1
      Contact( "T-06_ChiliFresh_1".IN_Dose_Header_1 )
      Contact( "IO_Valve_T06_FreshChili"."AV-06.12".FB_OPEN )
      wire#w2
      Coil( "T-06_ChiliFresh_1".IN_FBAV_Transfer )
   END_RUNG
   RUNG wire#w1
      Contact( "T-06_ChiliFresh_1".IN_Dose_Header_2 )
      Contact( "IO_Valve_T06_FreshChili"."AV-06.11".FB_OPEN )
   END_RUNG wire#w2
   RUNG wire#w1
      Contact( "IO_Valve_T05_Tomato"."AV-05.20".FB_OPEN )
      Contact( "IO_Valve_T06_FreshChili"."AV-06.02".FB_OPEN )
      Contact( "IO_Valve_T06_FreshChili"."AV-06.04".FB_OPEN )
      wire#w3
      Contact( "IO_Valve_T08_FreshChili"."AV-08.16".FB_OPEN )
      wire#w4
      Coil( "T-06_ChiliFresh_1".IN_FBAV_CIP_Tank )
   END_RUNG
   RUNG wire#w3
      Contact( "IO_Valve_T05_Tomato"."AV-05.14".FB_OPEN )
   END_RUNG wire#w4
   RUNG wire#w1
      Contact( "IO_Valve_T05_Tomato"."AV-05.20".FB_OPEN )
      Contact( "IO_Valve_T06_FreshChili"."AV-06.01".FB_OPEN )
      Contact( "IO_Valve_T06_FreshChili"."AV-06.05".FB_OPEN )
      wire#w5
      Contact( "IO_Valve_T06_FreshChili"."AV-06.13".FB_OPEN )
      wire#w6
      Coil( "T-06_ChiliFresh_1".IN_FBAV_CIP_Line )
   END_RUNG
   RUNG wire#w5
      Contact( "IO_Valve_T06_FreshChili"."AV-06.10".FB_OPEN )
   END_RUNG wire#w6
   RUNG wire#w1
      Contact( "T-06_ChiliFresh_1".Out_P_Inload )
      Coil( "T-06_ChiliFresh_1".IN_FBP_Inload )
   END_RUNG
   RUNG wire#w1
      Move(in := 0.0, out1 => "T-06_ChiliFresh_1".IN_FBP_Inload_SP)
   END_RUNG
   RUNG wire#w1
      Contact( "IO Motor MCC Preparation_DB"."P-06.01".QRUN )
      Coil( "T-06_ChiliFresh_1".IN_FBP_Transfer )
   END_RUNG
   RUNG wire#w1
      Move(in := "IO Motor MCC Preparation_DB"."P-06.01".QAct_Speed, out1 => "T-06_ChiliFresh_1".IN_FBP_Transfer_SP)
   END_RUNG
   RUNG wire#w1
      Contact( "IO Motor MCC Preparation_DB"."P-08.02".QRUN )
      Coil( "T-06_ChiliFresh_1".IN_FBP_CIP )
   END_RUNG
   RUNG wire#w1
      Move(in := "IO Motor MCC Preparation_DB"."P-08.02".QAct_Speed, out1 => "T-06_ChiliFresh_1".IN_FBP_CIP_Sp)
   END_RUNG
   // the same network as SCL:
   "T-06_ChiliFresh_1".IN_FBAV_Inload := "AlwaysTRUE" AND "T-06_ChiliFresh_1".Out_AV_Inload;
   "T-06_ChiliFresh_1".IN_FBAV_Outlet := "AlwaysTRUE" AND "IO_Valve_T06_FreshChili"."AV-06.03".FB_OPEN;
   "T-06_ChiliFresh_1".IN_FBAV_Transfer := "AlwaysTRUE" AND (("T-06_ChiliFresh_1".IN_Dose_Header_1 AND "IO_Valve_T06_FreshChili"."AV-06.12".FB_OPEN) OR ("T-06_ChiliFresh_1".IN_Dose_Header_2 AND "IO_Valve_T06_FreshChili"."AV-06.11".FB_OPEN));
   "T-06_ChiliFresh_1".IN_FBAV_CIP_Tank := "AlwaysTRUE" AND "IO_Valve_T05_Tomato"."AV-05.20".FB_OPEN AND "IO_Valve_T06_FreshChili"."AV-06.02".FB_OPEN AND "IO_Valve_T06_FreshChili"."AV-06.04".FB_OPEN AND ("IO_Valve_T08_FreshChili"."AV-08.16".FB_OPEN OR "IO_Valve_T05_Tomato"."AV-05.14".FB_OPEN);
   "T-06_ChiliFresh_1".IN_FBAV_CIP_Line := "AlwaysTRUE" AND "IO_Valve_T05_Tomato"."AV-05.20".FB_OPEN AND "IO_Valve_T06_FreshChili"."AV-06.01".FB_OPEN AND "IO_Valve_T06_FreshChili"."AV-06.05".FB_OPEN AND ("IO_Valve_T06_FreshChili"."AV-06.13".FB_OPEN OR "IO_Valve_T06_FreshChili"."AV-06.10".FB_OPEN);
   "T-06_ChiliFresh_1".IN_FBP_Inload := "AlwaysTRUE" AND "T-06_ChiliFresh_1".Out_P_Inload;
   IF "AlwaysTRUE" THEN "T-06_ChiliFresh_1".IN_FBP_Inload_SP := 0.0; END_IF;
   "T-06_ChiliFresh_1".IN_FBP_Transfer := "AlwaysTRUE" AND "IO Motor MCC Preparation_DB"."P-06.01".QRUN;
   IF "AlwaysTRUE" THEN
       "T-06_ChiliFresh_1".IN_FBP_Transfer_SP := "IO Motor MCC Preparation_DB"."P-06.01".QAct_Speed;
   END_IF;
   "T-06_ChiliFresh_1".IN_FBP_CIP := "AlwaysTRUE" AND "IO Motor MCC Preparation_DB"."P-08.02".QRUN;
   IF "AlwaysTRUE" THEN
       "T-06_ChiliFresh_1".IN_FBP_CIP_Sp := "IO Motor MCC Preparation_DB"."P-08.02".QAct_Speed;
   END_IF;
END_REGION

REGION Network 78: T-06.00 Comm to Blend
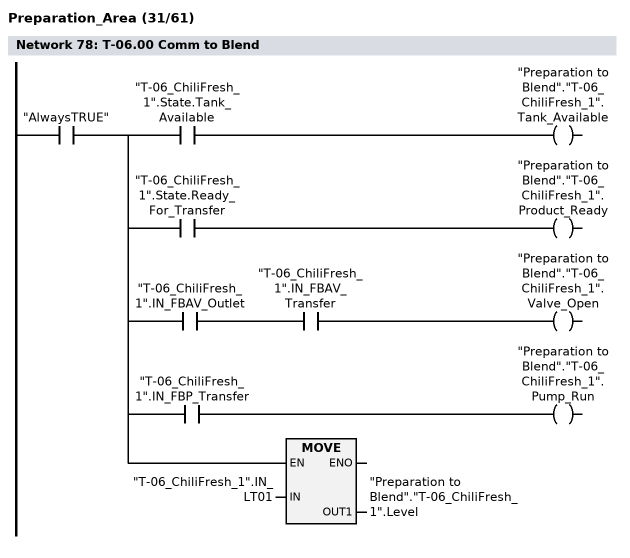
   RUNG wire#powerrail
      Contact( "AlwaysTRUE" )
      wire#w1
      Contact( "T-06_ChiliFresh_1".State.Tank_Available )
      Coil( "Preparation to Blend"."T-06_ChiliFresh_1".Tank_Available )
   END_RUNG
   RUNG wire#w1
      Contact( "T-06_ChiliFresh_1".State.Ready_For_Transfer )
      Coil( "Preparation to Blend"."T-06_ChiliFresh_1".Product_Ready )
   END_RUNG
   RUNG wire#w1
      Contact( "T-06_ChiliFresh_1".IN_FBAV_Outlet )
      Contact( "T-06_ChiliFresh_1".IN_FBAV_Transfer )
      Coil( "Preparation to Blend"."T-06_ChiliFresh_1".Valve_Open )
   END_RUNG
   RUNG wire#w1
      Contact( "T-06_ChiliFresh_1".IN_FBP_Transfer )
      Coil( "Preparation to Blend"."T-06_ChiliFresh_1".Pump_Run )
   END_RUNG
   RUNG wire#w1
      Move(in := "T-06_ChiliFresh_1".IN_LT01, out1 => "Preparation to Blend"."T-06_ChiliFresh_1".Level)
   END_RUNG
   // the same network as SCL:
   "Preparation to Blend"."T-06_ChiliFresh_1".Tank_Available := "AlwaysTRUE" AND "T-06_ChiliFresh_1".State.Tank_Available;
   "Preparation to Blend"."T-06_ChiliFresh_1".Product_Ready := "AlwaysTRUE" AND "T-06_ChiliFresh_1".State.Ready_For_Transfer;
   "Preparation to Blend"."T-06_ChiliFresh_1".Valve_Open := "AlwaysTRUE" AND "T-06_ChiliFresh_1".IN_FBAV_Outlet AND "T-06_ChiliFresh_1".IN_FBAV_Transfer;
   "Preparation to Blend"."T-06_ChiliFresh_1".Pump_Run := "AlwaysTRUE" AND "T-06_ChiliFresh_1".IN_FBP_Transfer;
   IF "AlwaysTRUE" THEN
       "Preparation to Blend"."T-06_ChiliFresh_1".Level := "T-06_ChiliFresh_1".IN_LT01;
   END_IF;
END_REGION

NETWORK
TITLE = T-07.00 DOSE ON OFF
      O     "Blend to Preparation"."T-20".Raw_Material.ChiliFresh_2.DoseRun;
      O     "Blend to Preparation"."T-21".Raw_Material.ChiliFresh_2.DoseRun;
      O     "Blend to Preparation"."T-30".Raw_Material.ChiliFresh_2.DoseRun;
      O     "Blend to Preparation"."T-31".Raw_Material.ChiliFresh_2.DoseRun;
      O     "Blend to Preparation"."T-40".Raw_Material.ChiliFresh_2.DoseRun;
      O     "Blend to Preparation"."T-41".Raw_Material.ChiliFresh_2.DoseRun;
      =     "T-07_ChiliFresh_2".IN_Dose_Run;

NETWORK
TITLE = T-07.00 DOSE PAUSE
      O     "Blend to Preparation"."T-20".Raw_Material.ChiliFresh_2.DoseHeld;
      O     "Blend to Preparation"."T-21".Raw_Material.ChiliFresh_2.DoseHeld;
      O     "Blend to Preparation"."T-30".Raw_Material.ChiliFresh_2.DoseHeld;
      O     "Blend to Preparation"."T-31".Raw_Material.ChiliFresh_2.DoseHeld;
      O     "Blend to Preparation"."T-40".Raw_Material.ChiliFresh_2.DoseHeld;
      O     "Blend to Preparation"."T-41".Raw_Material.ChiliFresh_2.DoseHeld;
      =     "T-07_ChiliFresh_2".IN_Dose_Held;

NETWORK
TITLE = T-07.00 DOSE VALVE CMD
      O(;
      A     "Blend to Preparation"."T-20".Raw_Material.ChiliFresh_2.DoseRun;
      A     "Blend to Preparation"."T-20".Raw_Material.ChiliFresh_2.ValveCMD;
      );
      O(;
      A     "Blend to Preparation"."T-21".Raw_Material.ChiliFresh_2.DoseRun;
      A     "Blend to Preparation"."T-21".Raw_Material.ChiliFresh_2.ValveCMD;
      );
      O(;
      A     "Blend to Preparation"."T-30".Raw_Material.ChiliFresh_2.DoseRun;
      A     "Blend to Preparation"."T-30".Raw_Material.ChiliFresh_2.ValveCMD;
      );
      O(;
      A     "Blend to Preparation"."T-31".Raw_Material.ChiliFresh_2.DoseRun;
      A     "Blend to Preparation"."T-31".Raw_Material.ChiliFresh_2.ValveCMD;
      );
      O(;
      A     "Blend to Preparation"."T-40".Raw_Material.ChiliFresh_2.DoseRun;
      A     "Blend to Preparation"."T-40".Raw_Material.ChiliFresh_2.ValveCMD;
      );
      O(;
      A     "Blend to Preparation"."T-41".Raw_Material.ChiliFresh_2.DoseRun;
      A     "Blend to Preparation"."T-41".Raw_Material.ChiliFresh_2.ValveCMD;
      );
      =     "T-07_ChiliFresh_2".IN_Dose_Valve_Cmd;



NETWORK
TITLE = T-07.00 DOSE Pump CMD
      O(;
      A     "Blend to Preparation"."T-20".Raw_Material.ChiliFresh_2.DoseRun;
      A     "Blend to Preparation"."T-20".Raw_Material.ChiliFresh_2.PumpCMD;
      );
      O(;
      A     "Blend to Preparation"."T-21".Raw_Material.ChiliFresh_2.DoseRun;
      A     "Blend to Preparation"."T-21".Raw_Material.ChiliFresh_2.PumpCMD;
      );
      O(;
      A     "Blend to Preparation"."T-30".Raw_Material.ChiliFresh_2.DoseRun;
      A     "Blend to Preparation"."T-30".Raw_Material.ChiliFresh_2.PumpCMD;
      );
      O(;
      A     "Blend to Preparation"."T-31".Raw_Material.ChiliFresh_2.DoseRun;
      A     "Blend to Preparation"."T-31".Raw_Material.ChiliFresh_2.PumpCMD;
      );
      O(;
      A     "Blend to Preparation"."T-40".Raw_Material.ChiliFresh_2.DoseRun;
      A     "Blend to Preparation"."T-40".Raw_Material.ChiliFresh_2.PumpCMD;
      );
      O(;
      A     "Blend to Preparation"."T-41".Raw_Material.ChiliFresh_2.DoseRun;
      A     "Blend to Preparation"."T-41".Raw_Material.ChiliFresh_2.PumpCMD;
      );
      =     "T-07_ChiliFresh_2".IN_Dose_Pump_Cmd;



NETWORK
TITLE = T-07.00 DOSE PUMP SPEED
// Checking
      O     "Blend to Preparation"."T-20".Raw_Material.ChiliFresh_2.DoseRun;
      JC    SP_07_FROM_20;
      O     "Blend to Preparation"."T-21".Raw_Material.ChiliFresh_2.DoseRun;
      JC    SP_07_FROM_21;
      O     "Blend to Preparation"."T-30".Raw_Material.ChiliFresh_2.DoseRun;
      JC    SP_07_FROM_30;
      O     "Blend to Preparation"."T-31".Raw_Material.ChiliFresh_2.DoseRun;
      JC    SP_07_FROM_31;
      O     "Blend to Preparation"."T-40".Raw_Material.ChiliFresh_2.DoseRun;
      JC    SP_07_FROM_40;
      O     "Blend to Preparation"."T-41".Raw_Material.ChiliFresh_2.DoseRun;
      JC    SP_07_FROM_41;
//Jump to end if Blend not Dosing
      JC    SP_07_SELF;
//Load Set Point
SP_07_FROM_20:L     "Blend to Preparation".Recipe."T-20".ChiliFresh_2.SP_PumpSpeed;
      T     "T-07_ChiliFresh_2".IN_Dose_Pump_Sp;
      JC    SP_07_SELF;
SP_07_FROM_21:L     "Blend to Preparation".Recipe."T-21".ChiliFresh_2.SP_PumpSpeed;
      T     "T-07_ChiliFresh_2".IN_Dose_Pump_Sp;
      JC    SP_07_SELF;
SP_07_FROM_30:L     "Blend to Preparation".Recipe."T-30".ChiliFresh_2.SP_PumpSpeed;
      T     "T-07_ChiliFresh_2".IN_Dose_Pump_Sp;
      JC    SP_07_SELF;
SP_07_FROM_31:L     "Blend to Preparation".Recipe."T-31".ChiliFresh_2.SP_PumpSpeed;
      T     "T-07_ChiliFresh_2".IN_Dose_Pump_Sp;
      JC    SP_07_SELF;
SP_07_FROM_40:L     "Blend to Preparation".Recipe."T-40".ChiliFresh_2.SP_PumpSpeed;
      T     "T-07_ChiliFresh_2".IN_Dose_Pump_Sp;
      JC    SP_07_SELF;
SP_07_FROM_41:L     "Blend to Preparation".Recipe."T-41".ChiliFresh_2.SP_PumpSpeed;
      T     "T-07_ChiliFresh_2".IN_Dose_Pump_Sp;
      JC    SP_07_SELF;
// END
SP_07_SELF:L     "T-07_ChiliFresh_2".IN_Dose_Pump_Sp;
      T     "T-07_ChiliFresh_2".IN_Dose_Pump_Sp;


NETWORK
TITLE = T-07.00 Header Req
// HEADER 1 Req
      O     "Blend to Preparation"."T-20".Raw_Material.ChiliFresh_2.Header1_Req;
      O     "Blend to Preparation"."T-21".Raw_Material.ChiliFresh_2.Header1_Req;
      O     "Blend to Preparation"."T-30".Raw_Material.ChiliFresh_2.Header1_Req;
      O     "Blend to Preparation"."T-31".Raw_Material.ChiliFresh_2.Header1_Req;
      O     "Blend to Preparation"."T-40".Raw_Material.ChiliFresh_2.Header1_Req;
      O     "Blend to Preparation"."T-41".Raw_Material.ChiliFresh_2.Header1_Req;
      =     "T-07_ChiliFresh_2".IN_Dose_Header_1;

// HEADER 2 Req
      O     "Blend to Preparation"."T-20".Raw_Material.ChiliFresh_2.Header2_Req;
      O     "Blend to Preparation"."T-21".Raw_Material.ChiliFresh_2.Header2_Req;
      O     "Blend to Preparation"."T-30".Raw_Material.ChiliFresh_2.Header2_Req;
      O     "Blend to Preparation"."T-31".Raw_Material.ChiliFresh_2.Header2_Req;
      O     "Blend to Preparation"."T-40".Raw_Material.ChiliFresh_2.Header2_Req;
      O     "Blend to Preparation"."T-41".Raw_Material.ChiliFresh_2.Header2_Req;
      =     "T-07_ChiliFresh_2".IN_Dose_Header_2;


REGION Network 87: T-07.00 LineTransferOK
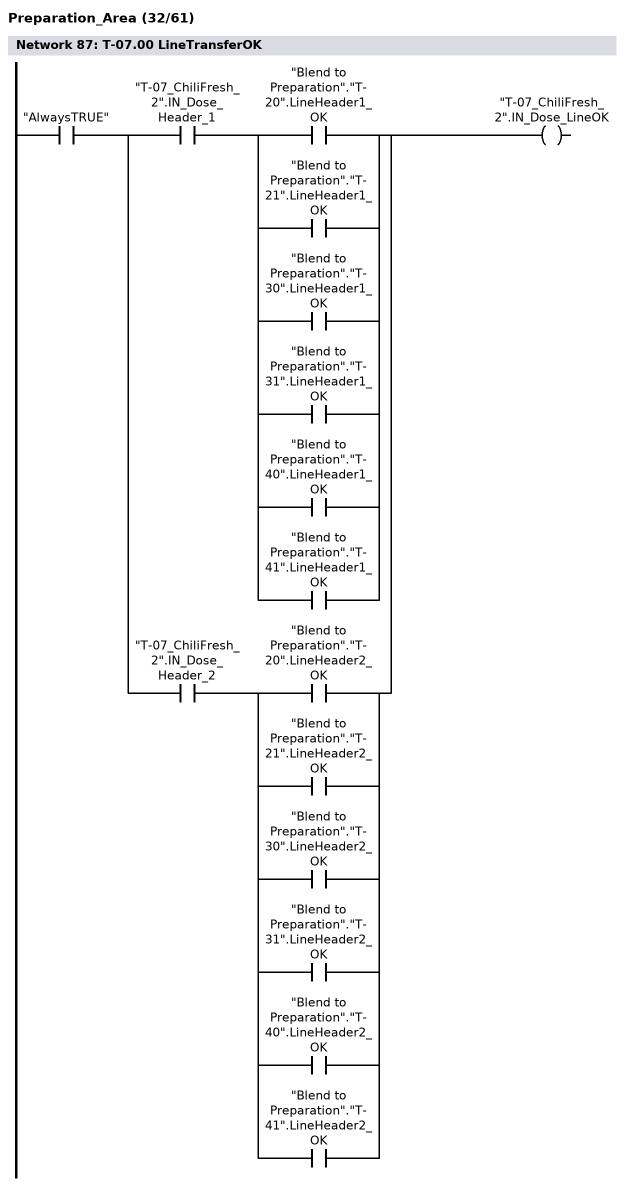
   RUNG wire#powerrail
      Contact( "AlwaysTRUE" )
      wire#w1
      Contact( "T-07_ChiliFresh_2".IN_Dose_Header_1 )
      wire#w2
      Contact( "Blend to Preparation"."T-20".LineHeader1_OK )
      wire#w3
      Coil( "T-07_ChiliFresh_2".IN_Dose_LineOK )
   END_RUNG
   RUNG wire#w2
      Contact( "Blend to Preparation"."T-21".LineHeader1_OK )
   END_RUNG wire#w3
   RUNG wire#w2
      Contact( "Blend to Preparation"."T-30".LineHeader1_OK )
   END_RUNG wire#w3
   RUNG wire#w2
      Contact( "Blend to Preparation"."T-31".LineHeader1_OK )
   END_RUNG wire#w3
   RUNG wire#w2
      Contact( "Blend to Preparation"."T-40".LineHeader1_OK )
   END_RUNG wire#w3
   RUNG wire#w2
      Contact( "Blend to Preparation"."T-41".LineHeader1_OK )
   END_RUNG wire#w3
   RUNG wire#w1
      Contact( "T-07_ChiliFresh_2".IN_Dose_Header_2 )
      wire#w4
      Contact( "Blend to Preparation"."T-20".LineHeader2_OK )
   END_RUNG wire#w3
   RUNG wire#w4
      Contact( "Blend to Preparation"."T-21".LineHeader2_OK )
   END_RUNG wire#w3
   RUNG wire#w4
      Contact( "Blend to Preparation"."T-30".LineHeader2_OK )
   END_RUNG wire#w3
   RUNG wire#w4
      Contact( "Blend to Preparation"."T-31".LineHeader2_OK )
   END_RUNG wire#w3
   RUNG wire#w4
      Contact( "Blend to Preparation"."T-40".LineHeader2_OK )
   END_RUNG wire#w3
   RUNG wire#w4
      Contact( "Blend to Preparation"."T-41".LineHeader2_OK )
   END_RUNG wire#w3
   // the same network as SCL:
   "T-07_ChiliFresh_2".IN_Dose_LineOK := "AlwaysTRUE" AND (("T-07_ChiliFresh_2".IN_Dose_Header_1 AND ("Blend to Preparation"."T-20".LineHeader1_OK OR "Blend to Preparation"."T-21".LineHeader1_OK OR "Blend to Preparation"."T-30".LineHeader1_OK OR "Blend to Preparation"."T-31".LineHeader1_OK OR "Blend to Preparation"."T-40".LineHeader1_OK OR "Blend to Preparation"."T-41".LineHeader1_OK)) OR ("T-07_ChiliFresh_2".IN_Dose_Header_2 AND ("Blend to Preparation"."T-20".LineHeader2_OK OR "Blend to Preparation"."T-21".LineHeader2_OK OR "Blend to Preparation"."T-30".LineHeader2_OK OR "Blend to Preparation"."T-31".LineHeader2_OK OR "Blend to Preparation"."T-40".LineHeader2_OK OR "Blend to Preparation"."T-41".LineHeader2_OK)));
END_REGION

REGION Network 88: T-07____Chili Fresh 2
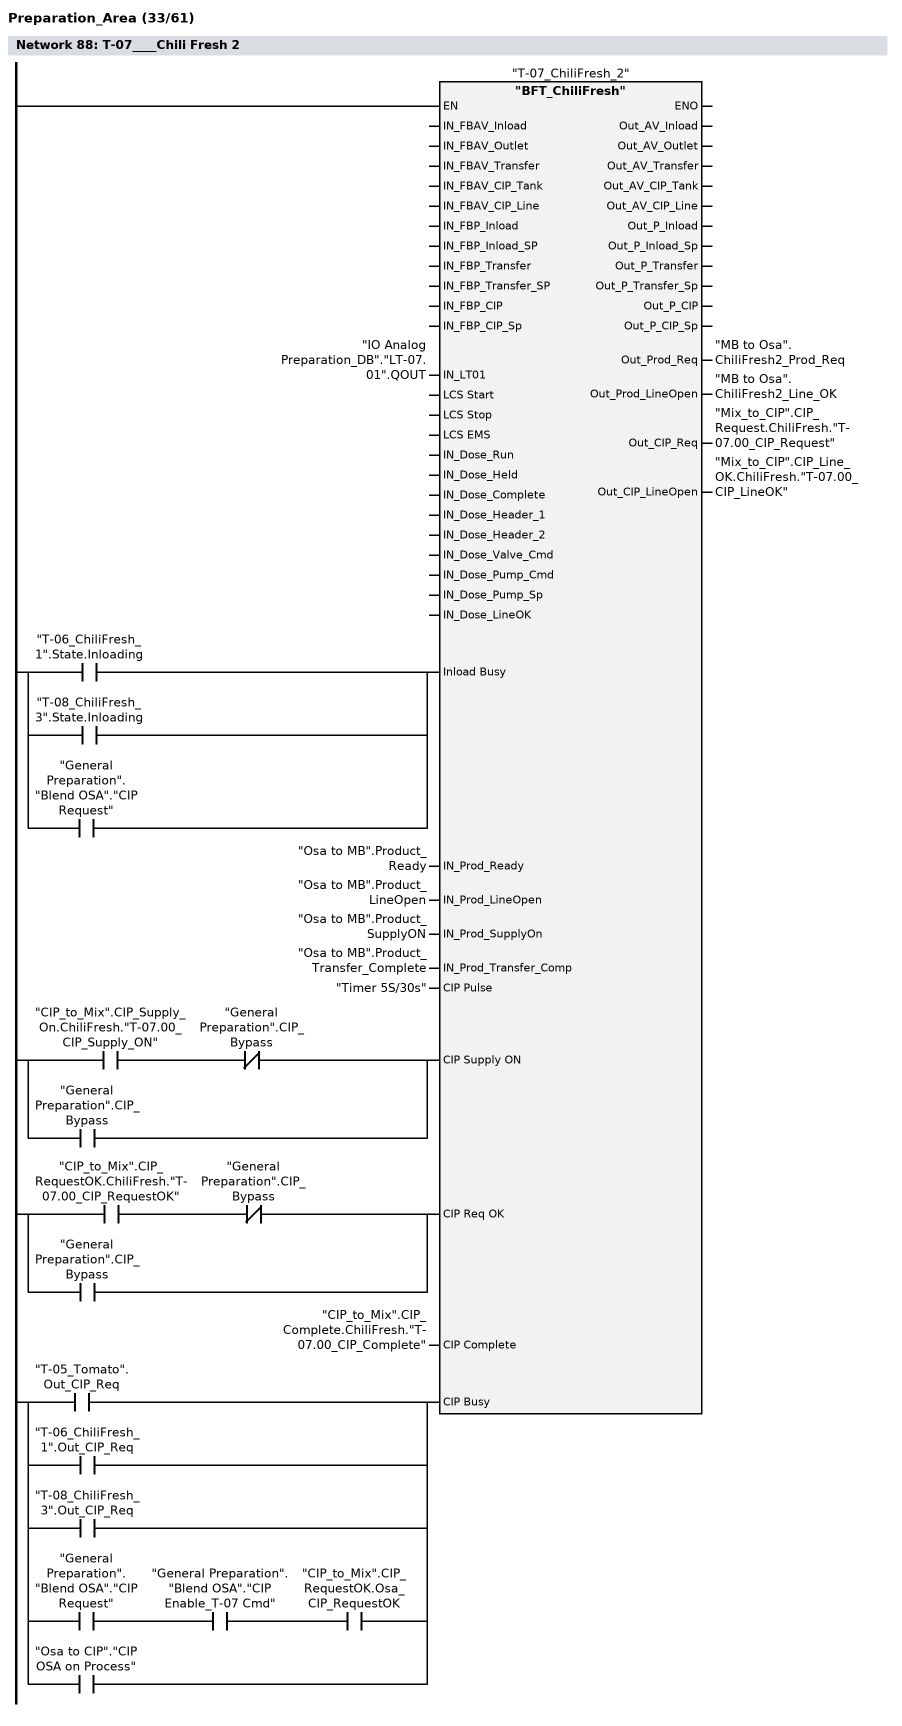
   RUNG wire#powerrail
      "T-07_ChiliFresh_2"("Inload Busy" := wire#w1, "CIP Supply ON" := wire#w2, "CIP Req OK" := wire#w3, "CIP Busy" := wire#w4, IN_FBAV_Inload :=, IN_FBAV_Outlet :=, IN_FBAV_Transfer :=, IN_FBAV_CIP_Tank :=, IN_FBAV_CIP_Line :=, IN_FBP_Inload :=, IN_FBP_Inload_SP :=, IN_FBP_Transfer :=, IN_FBP_Transfer_SP :=, IN_FBP_CIP :=, IN_FBP_CIP_Sp :=, IN_LT01 := "IO Analog Preparation_DB"."LT-07.01".QOUT, "LCS Start" :=, "LCS Stop" :=, "LCS EMS" :=, IN_Dose_Run :=, IN_Dose_Held :=, IN_Dose_Complete :=, IN_Dose_Header_1 :=, IN_Dose_Header_2 :=, IN_Dose_Valve_Cmd :=, IN_Dose_Pump_Cmd :=, IN_Dose_Pump_Sp :=, IN_Dose_LineOK :=, IN_Prod_Ready := "Osa to MB".Product_Ready, IN_Prod_LineOpen := "Osa to MB".Product_LineOpen, IN_Prod_SupplyOn := "Osa to MB".Product_SupplyON, IN_Prod_Transfer_Comp := "Osa to MB".Product_Transfer_Complete, "CIP Pulse" := "Timer 5S/30s", "CIP Complete" := "CIP_to_Mix".CIP_Complete.ChiliFresh."T-07.00_CIP_Complete", Out_AV_Inload =>, Out_AV_Outlet =>, Out_AV_Transfer =>, Out_AV_CIP_Tank =>, Out_AV_CIP_Line =>, Out_P_Inload =>, Out_P_Inload_Sp =>, Out_P_Transfer =>, Out_P_Transfer_Sp =>, Out_P_CIP =>, Out_P_CIP_Sp =>, Out_Prod_Req => "MB to Osa".ChiliFresh2_Prod_Req, Out_Prod_LineOpen => "MB to Osa".ChiliFresh2_Line_OK, Out_CIP_Req => "Mix_to_CIP".CIP_Request.ChiliFresh."T-07.00_CIP_Request", Out_CIP_LineOpen => "Mix_to_CIP".CIP_Line_OK.ChiliFresh."T-07.00_CIP_LineOK")
   END_RUNG
   RUNG wire#powerrail
      Contact( "T-06_ChiliFresh_1".State.Inloading )
   END_RUNG wire#w1
   RUNG wire#powerrail
      Contact( "T-08_ChiliFresh_3".State.Inloading )
   END_RUNG wire#w1
   RUNG wire#powerrail
      Contact( "General Preparation"."Blend OSA"."CIP Request" )
   END_RUNG wire#w1
   RUNG wire#powerrail
      Contact( "CIP_to_Mix".CIP_Supply_On.ChiliFresh."T-07.00_CIP_Supply_ON" )
      I_Contact( "General Preparation".CIP_Bypass )
   END_RUNG wire#w2
   RUNG wire#powerrail
      Contact( "General Preparation".CIP_Bypass )
   END_RUNG wire#w2
   RUNG wire#powerrail
      Contact( "CIP_to_Mix".CIP_RequestOK.ChiliFresh."T-07.00_CIP_RequestOK" )
      I_Contact( "General Preparation".CIP_Bypass )
   END_RUNG wire#w3
   RUNG wire#powerrail
      Contact( "General Preparation".CIP_Bypass )
   END_RUNG wire#w3
   RUNG wire#powerrail
      Contact( "T-05_Tomato".Out_CIP_Req )
   END_RUNG wire#w4
   RUNG wire#powerrail
      Contact( "T-06_ChiliFresh_1".Out_CIP_Req )
   END_RUNG wire#w4
   RUNG wire#powerrail
      Contact( "T-08_ChiliFresh_3".Out_CIP_Req )
   END_RUNG wire#w4
   RUNG wire#powerrail
      Contact( "General Preparation"."Blend OSA"."CIP Request" )
      Contact( "General Preparation"."Blend OSA"."CIP Enable_T-07 Cmd" )
      Contact( "CIP_to_Mix".CIP_RequestOK.Osa_CIP_RequestOK )
   END_RUNG wire#w4
   RUNG wire#powerrail
      Contact( "Osa to CIP"."CIP OSA on Process" )
   END_RUNG wire#w4
   // the same network as SCL:
   "T-07_ChiliFresh_2"(IN_LT01 := "IO Analog Preparation_DB"."LT-07.01".QOUT,   // "BFT_ChiliFresh"
                       "Inload Busy" := "T-06_ChiliFresh_1".State.Inloading OR "T-08_ChiliFresh_3".State.Inloading OR "General Preparation"."Blend OSA"."CIP Request",
                       IN_Prod_Ready := "Osa to MB".Product_Ready,
                       IN_Prod_LineOpen := "Osa to MB".Product_LineOpen,
                       IN_Prod_SupplyOn := "Osa to MB".Product_SupplyON,
                       IN_Prod_Transfer_Comp := "Osa to MB".Product_Transfer_Complete,
                       "CIP Pulse" := "Timer 5S/30s",
                       "CIP Supply ON" := ("CIP_to_Mix".CIP_Supply_On.ChiliFresh."T-07.00_CIP_Supply_ON" AND NOT "General Preparation".CIP_Bypass) OR "General Preparation".CIP_Bypass,
                       "CIP Req OK" := ("CIP_to_Mix".CIP_RequestOK.ChiliFresh."T-07.00_CIP_RequestOK" AND NOT "General Preparation".CIP_Bypass) OR "General Preparation".CIP_Bypass,
                       "CIP Complete" := "CIP_to_Mix".CIP_Complete.ChiliFresh."T-07.00_CIP_Complete",
                       "CIP Busy" := "T-05_Tomato".Out_CIP_Req OR "T-06_ChiliFresh_1".Out_CIP_Req OR "T-08_ChiliFresh_3".Out_CIP_Req OR ("General Preparation"."Blend OSA"."CIP Request" AND "General Preparation"."Blend OSA"."CIP Enable_T-07 Cmd" AND "CIP_to_Mix".CIP_RequestOK.Osa_CIP_RequestOK) OR "Osa to CIP"."CIP OSA on Process",
                       Out_Prod_Req => "MB to Osa".ChiliFresh2_Prod_Req,
                       Out_Prod_LineOpen => "MB to Osa".ChiliFresh2_Line_OK,
                       Out_CIP_Req => "Mix_to_CIP".CIP_Request.ChiliFresh."T-07.00_CIP_Request",
                       Out_CIP_LineOpen => "Mix_to_CIP".CIP_Line_OK.ChiliFresh."T-07.00_CIP_LineOK");
END_REGION

REGION Network 89: T-07.00 Valve Cmd
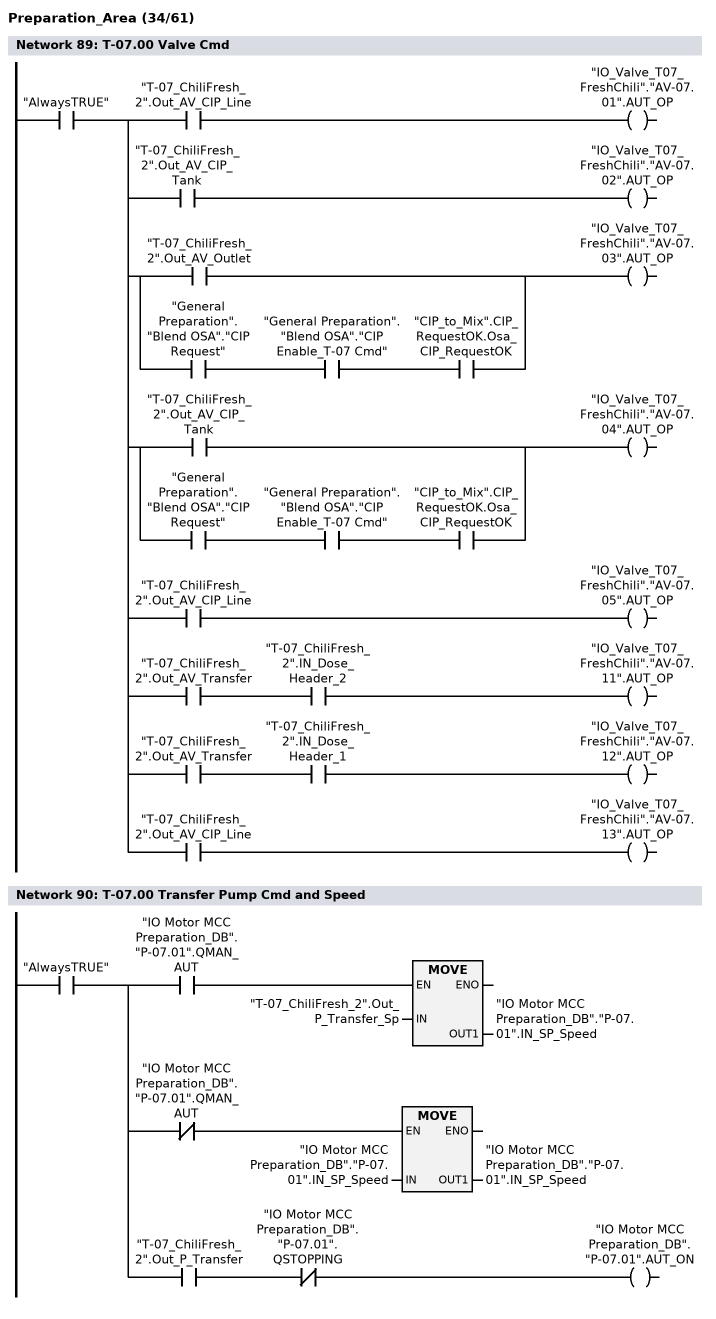
   RUNG wire#powerrail
      Contact( "AlwaysTRUE" )
      wire#w1
      Contact( "T-07_ChiliFresh_2".Out_AV_CIP_Line )
      Coil( "IO_Valve_T07_FreshChili"."AV-07.01".AUT_OP )
   END_RUNG
   RUNG wire#w1
      Contact( "T-07_ChiliFresh_2".Out_AV_CIP_Tank )
      Coil( "IO_Valve_T07_FreshChili"."AV-07.02".AUT_OP )
   END_RUNG
   RUNG wire#w1
      Contact( "T-07_ChiliFresh_2".Out_AV_Outlet )
      wire#w2
      Coil( "IO_Valve_T07_FreshChili"."AV-07.03".AUT_OP )
   END_RUNG
   RUNG wire#w1
      Contact( "General Preparation"."Blend OSA"."CIP Request" )
      Contact( "General Preparation"."Blend OSA"."CIP Enable_T-07 Cmd" )
      Contact( "CIP_to_Mix".CIP_RequestOK.Osa_CIP_RequestOK )
   END_RUNG wire#w2
   RUNG wire#w1
      Contact( "T-07_ChiliFresh_2".Out_AV_CIP_Tank )
      wire#w3
      Coil( "IO_Valve_T07_FreshChili"."AV-07.04".AUT_OP )
   END_RUNG
   RUNG wire#w1
      Contact( "General Preparation"."Blend OSA"."CIP Request" )
      Contact( "General Preparation"."Blend OSA"."CIP Enable_T-07 Cmd" )
      Contact( "CIP_to_Mix".CIP_RequestOK.Osa_CIP_RequestOK )
   END_RUNG wire#w3
   RUNG wire#w1
      Contact( "T-07_ChiliFresh_2".Out_AV_CIP_Line )
      Coil( "IO_Valve_T07_FreshChili"."AV-07.05".AUT_OP )
   END_RUNG
   RUNG wire#w1
      Contact( "T-07_ChiliFresh_2".Out_AV_Transfer )
      Contact( "T-07_ChiliFresh_2".IN_Dose_Header_2 )
      Coil( "IO_Valve_T07_FreshChili"."AV-07.11".AUT_OP )
   END_RUNG
   RUNG wire#w1
      Contact( "T-07_ChiliFresh_2".Out_AV_Transfer )
      Contact( "T-07_ChiliFresh_2".IN_Dose_Header_1 )
      Coil( "IO_Valve_T07_FreshChili"."AV-07.12".AUT_OP )
   END_RUNG
   RUNG wire#w1
      Contact( "T-07_ChiliFresh_2".Out_AV_CIP_Line )
      Coil( "IO_Valve_T07_FreshChili"."AV-07.13".AUT_OP )
   END_RUNG
   // the same network as SCL:
   "IO_Valve_T07_FreshChili"."AV-07.01".AUT_OP := "AlwaysTRUE" AND "T-07_ChiliFresh_2".Out_AV_CIP_Line;
   "IO_Valve_T07_FreshChili"."AV-07.02".AUT_OP := "AlwaysTRUE" AND "T-07_ChiliFresh_2".Out_AV_CIP_Tank;
   "IO_Valve_T07_FreshChili"."AV-07.03".AUT_OP := "AlwaysTRUE" AND ("T-07_ChiliFresh_2".Out_AV_Outlet OR ("General Preparation"."Blend OSA"."CIP Request" AND "General Preparation"."Blend OSA"."CIP Enable_T-07 Cmd" AND "CIP_to_Mix".CIP_RequestOK.Osa_CIP_RequestOK));
   "IO_Valve_T07_FreshChili"."AV-07.04".AUT_OP := "AlwaysTRUE" AND ("T-07_ChiliFresh_2".Out_AV_CIP_Tank OR ("General Preparation"."Blend OSA"."CIP Request" AND "General Preparation"."Blend OSA"."CIP Enable_T-07 Cmd" AND "CIP_to_Mix".CIP_RequestOK.Osa_CIP_RequestOK));
   "IO_Valve_T07_FreshChili"."AV-07.05".AUT_OP := "AlwaysTRUE" AND "T-07_ChiliFresh_2".Out_AV_CIP_Line;
   "IO_Valve_T07_FreshChili"."AV-07.11".AUT_OP := "AlwaysTRUE" AND "T-07_ChiliFresh_2".Out_AV_Transfer AND "T-07_ChiliFresh_2".IN_Dose_Header_2;
   "IO_Valve_T07_FreshChili"."AV-07.12".AUT_OP := "AlwaysTRUE" AND "T-07_ChiliFresh_2".Out_AV_Transfer AND "T-07_ChiliFresh_2".IN_Dose_Header_1;
   "IO_Valve_T07_FreshChili"."AV-07.13".AUT_OP := "AlwaysTRUE" AND "T-07_ChiliFresh_2".Out_AV_CIP_Line;
END_REGION

REGION Network 90: T-07.00 Transfer Pump Cmd and Speed
   RUNG wire#powerrail
      Contact( "AlwaysTRUE" )
      wire#w1
      Contact( "IO Motor MCC Preparation_DB"."P-07.01".QMAN_AUT )
      Move(in := "T-07_ChiliFresh_2".Out_P_Transfer_Sp, out1 => "IO Motor MCC Preparation_DB"."P-07.01".IN_SP_Speed)
   END_RUNG
   RUNG wire#w1
      I_Contact( "IO Motor MCC Preparation_DB"."P-07.01".QMAN_AUT )
      Move(in := "IO Motor MCC Preparation_DB"."P-07.01".IN_SP_Speed, out1 => "IO Motor MCC Preparation_DB"."P-07.01".IN_SP_Speed)
   END_RUNG
   RUNG wire#w1
      Contact( "T-07_ChiliFresh_2".Out_P_Transfer )
      I_Contact( "IO Motor MCC Preparation_DB"."P-07.01".QSTOPPING )
      Coil( "IO Motor MCC Preparation_DB"."P-07.01".AUT_ON )
   END_RUNG
   // the same network as SCL:
   IF "AlwaysTRUE" AND "IO Motor MCC Preparation_DB"."P-07.01".QMAN_AUT THEN
       "IO Motor MCC Preparation_DB"."P-07.01".IN_SP_Speed := "T-07_ChiliFresh_2".Out_P_Transfer_Sp;
   END_IF;
   IF "AlwaysTRUE" AND NOT "IO Motor MCC Preparation_DB"."P-07.01".QMAN_AUT THEN
       "IO Motor MCC Preparation_DB"."P-07.01".IN_SP_Speed := "IO Motor MCC Preparation_DB"."P-07.01".IN_SP_Speed;
   END_IF;
   "IO Motor MCC Preparation_DB"."P-07.01".AUT_ON := "AlwaysTRUE" AND "T-07_ChiliFresh_2".Out_P_Transfer AND NOT "IO Motor MCC Preparation_DB"."P-07.01".QSTOPPING;
END_REGION

REGION Network 91: T-07.00 Feedback Instrument
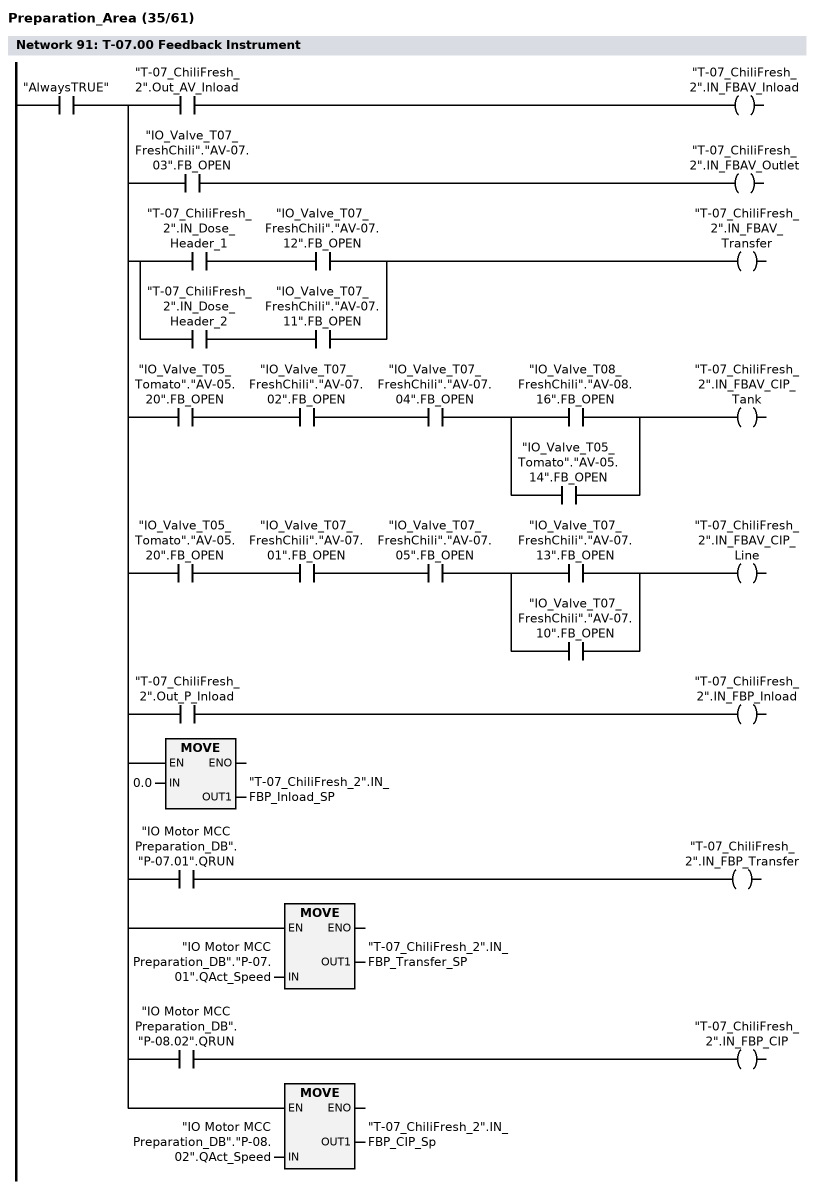
   RUNG wire#powerrail
      Contact( "AlwaysTRUE" )
      wire#w1
      Contact( "T-07_ChiliFresh_2".Out_AV_Inload )
      Coil( "T-07_ChiliFresh_2".IN_FBAV_Inload )
   END_RUNG
   RUNG wire#w1
      Contact( "IO_Valve_T07_FreshChili"."AV-07.03".FB_OPEN )
      Coil( "T-07_ChiliFresh_2".IN_FBAV_Outlet )
   END_RUNG
   RUNG wire#w1
      Contact( "T-07_ChiliFresh_2".IN_Dose_Header_1 )
      Contact( "IO_Valve_T07_FreshChili"."AV-07.12".FB_OPEN )
      wire#w2
      Coil( "T-07_ChiliFresh_2".IN_FBAV_Transfer )
   END_RUNG
   RUNG wire#w1
      Contact( "T-07_ChiliFresh_2".IN_Dose_Header_2 )
      Contact( "IO_Valve_T07_FreshChili"."AV-07.11".FB_OPEN )
   END_RUNG wire#w2
   RUNG wire#w1
      Contact( "IO_Valve_T05_Tomato"."AV-05.20".FB_OPEN )
      Contact( "IO_Valve_T07_FreshChili"."AV-07.02".FB_OPEN )
      Contact( "IO_Valve_T07_FreshChili"."AV-07.04".FB_OPEN )
      wire#w3
      Contact( "IO_Valve_T08_FreshChili"."AV-08.16".FB_OPEN )
      wire#w4
      Coil( "T-07_ChiliFresh_2".IN_FBAV_CIP_Tank )
   END_RUNG
   RUNG wire#w3
      Contact( "IO_Valve_T05_Tomato"."AV-05.14".FB_OPEN )
   END_RUNG wire#w4
   RUNG wire#w1
      Contact( "IO_Valve_T05_Tomato"."AV-05.20".FB_OPEN )
      Contact( "IO_Valve_T07_FreshChili"."AV-07.01".FB_OPEN )
      Contact( "IO_Valve_T07_FreshChili"."AV-07.05".FB_OPEN )
      wire#w5
      Contact( "IO_Valve_T07_FreshChili"."AV-07.13".FB_OPEN )
      wire#w6
      Coil( "T-07_ChiliFresh_2".IN_FBAV_CIP_Line )
   END_RUNG
   RUNG wire#w5
      Contact( "IO_Valve_T07_FreshChili"."AV-07.10".FB_OPEN )
   END_RUNG wire#w6
   RUNG wire#w1
      Contact( "T-07_ChiliFresh_2".Out_P_Inload )
      Coil( "T-07_ChiliFresh_2".IN_FBP_Inload )
   END_RUNG
   RUNG wire#w1
      Move(in := 0.0, out1 => "T-07_ChiliFresh_2".IN_FBP_Inload_SP)
   END_RUNG
   RUNG wire#w1
      Contact( "IO Motor MCC Preparation_DB"."P-07.01".QRUN )
      Coil( "T-07_ChiliFresh_2".IN_FBP_Transfer )
   END_RUNG
   RUNG wire#w1
      Move(in := "IO Motor MCC Preparation_DB"."P-07.01".QAct_Speed, out1 => "T-07_ChiliFresh_2".IN_FBP_Transfer_SP)
   END_RUNG
   RUNG wire#w1
      Contact( "IO Motor MCC Preparation_DB"."P-08.02".QRUN )
      Coil( "T-07_ChiliFresh_2".IN_FBP_CIP )
   END_RUNG
   RUNG wire#w1
      Move(in := "IO Motor MCC Preparation_DB"."P-08.02".QAct_Speed, out1 => "T-07_ChiliFresh_2".IN_FBP_CIP_Sp)
   END_RUNG
   // the same network as SCL:
   "T-07_ChiliFresh_2".IN_FBAV_Inload := "AlwaysTRUE" AND "T-07_ChiliFresh_2".Out_AV_Inload;
   "T-07_ChiliFresh_2".IN_FBAV_Outlet := "AlwaysTRUE" AND "IO_Valve_T07_FreshChili"."AV-07.03".FB_OPEN;
   "T-07_ChiliFresh_2".IN_FBAV_Transfer := "AlwaysTRUE" AND (("T-07_ChiliFresh_2".IN_Dose_Header_1 AND "IO_Valve_T07_FreshChili"."AV-07.12".FB_OPEN) OR ("T-07_ChiliFresh_2".IN_Dose_Header_2 AND "IO_Valve_T07_FreshChili"."AV-07.11".FB_OPEN));
   "T-07_ChiliFresh_2".IN_FBAV_CIP_Tank := "AlwaysTRUE" AND "IO_Valve_T05_Tomato"."AV-05.20".FB_OPEN AND "IO_Valve_T07_FreshChili"."AV-07.02".FB_OPEN AND "IO_Valve_T07_FreshChili"."AV-07.04".FB_OPEN AND ("IO_Valve_T08_FreshChili"."AV-08.16".FB_OPEN OR "IO_Valve_T05_Tomato"."AV-05.14".FB_OPEN);
   "T-07_ChiliFresh_2".IN_FBAV_CIP_Line := "AlwaysTRUE" AND "IO_Valve_T05_Tomato"."AV-05.20".FB_OPEN AND "IO_Valve_T07_FreshChili"."AV-07.01".FB_OPEN AND "IO_Valve_T07_FreshChili"."AV-07.05".FB_OPEN AND ("IO_Valve_T07_FreshChili"."AV-07.13".FB_OPEN OR "IO_Valve_T07_FreshChili"."AV-07.10".FB_OPEN);
   "T-07_ChiliFresh_2".IN_FBP_Inload := "AlwaysTRUE" AND "T-07_ChiliFresh_2".Out_P_Inload;
   IF "AlwaysTRUE" THEN "T-07_ChiliFresh_2".IN_FBP_Inload_SP := 0.0; END_IF;
   "T-07_ChiliFresh_2".IN_FBP_Transfer := "AlwaysTRUE" AND "IO Motor MCC Preparation_DB"."P-07.01".QRUN;
   IF "AlwaysTRUE" THEN
       "T-07_ChiliFresh_2".IN_FBP_Transfer_SP := "IO Motor MCC Preparation_DB"."P-07.01".QAct_Speed;
   END_IF;
   "T-07_ChiliFresh_2".IN_FBP_CIP := "AlwaysTRUE" AND "IO Motor MCC Preparation_DB"."P-08.02".QRUN;
   IF "AlwaysTRUE" THEN
       "T-07_ChiliFresh_2".IN_FBP_CIP_Sp := "IO Motor MCC Preparation_DB"."P-08.02".QAct_Speed;
   END_IF;
END_REGION

REGION Network 92: T-07.00 Comm to Blend
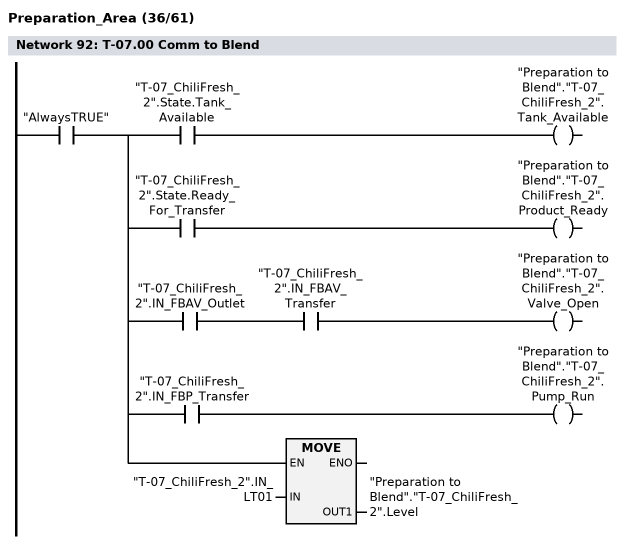
   RUNG wire#powerrail
      Contact( "AlwaysTRUE" )
      wire#w1
      Contact( "T-07_ChiliFresh_2".State.Tank_Available )
      Coil( "Preparation to Blend"."T-07_ChiliFresh_2".Tank_Available )
   END_RUNG
   RUNG wire#w1
      Contact( "T-07_ChiliFresh_2".State.Ready_For_Transfer )
      Coil( "Preparation to Blend"."T-07_ChiliFresh_2".Product_Ready )
   END_RUNG
   RUNG wire#w1
      Contact( "T-07_ChiliFresh_2".IN_FBAV_Outlet )
      Contact( "T-07_ChiliFresh_2".IN_FBAV_Transfer )
      Coil( "Preparation to Blend"."T-07_ChiliFresh_2".Valve_Open )
   END_RUNG
   RUNG wire#w1
      Contact( "T-07_ChiliFresh_2".IN_FBP_Transfer )
      Coil( "Preparation to Blend"."T-07_ChiliFresh_2".Pump_Run )
   END_RUNG
   RUNG wire#w1
      Move(in := "T-07_ChiliFresh_2".IN_LT01, out1 => "Preparation to Blend"."T-07_ChiliFresh_2".Level)
   END_RUNG
   // the same network as SCL:
   "Preparation to Blend"."T-07_ChiliFresh_2".Tank_Available := "AlwaysTRUE" AND "T-07_ChiliFresh_2".State.Tank_Available;
   "Preparation to Blend"."T-07_ChiliFresh_2".Product_Ready := "AlwaysTRUE" AND "T-07_ChiliFresh_2".State.Ready_For_Transfer;
   "Preparation to Blend"."T-07_ChiliFresh_2".Valve_Open := "AlwaysTRUE" AND "T-07_ChiliFresh_2".IN_FBAV_Outlet AND "T-07_ChiliFresh_2".IN_FBAV_Transfer;
   "Preparation to Blend"."T-07_ChiliFresh_2".Pump_Run := "AlwaysTRUE" AND "T-07_ChiliFresh_2".IN_FBP_Transfer;
   IF "AlwaysTRUE" THEN
       "Preparation to Blend"."T-07_ChiliFresh_2".Level := "T-07_ChiliFresh_2".IN_LT01;
   END_IF;
END_REGION

NETWORK
TITLE = T-08.00 DOSE ON OFF
      O     "Blend to Preparation"."T-20".Raw_Material.ChiliFresh_3.DoseRun;
      O     "Blend to Preparation"."T-21".Raw_Material.ChiliFresh_3.DoseRun;
      O     "Blend to Preparation"."T-30".Raw_Material.ChiliFresh_3.DoseRun;
      O     "Blend to Preparation"."T-31".Raw_Material.ChiliFresh_3.DoseRun;
      O     "Blend to Preparation"."T-40".Raw_Material.ChiliFresh_3.DoseRun;
      O     "Blend to Preparation"."T-41".Raw_Material.ChiliFresh_3.DoseRun;
      =     "T-08_ChiliFresh_3".IN_Dose_Run;

NETWORK
TITLE = T-08.00 DOSE PAUSE
      O     "Blend to Preparation"."T-20".Raw_Material.ChiliFresh_3.DoseHeld;
      O     "Blend to Preparation"."T-21".Raw_Material.ChiliFresh_3.DoseHeld;
      O     "Blend to Preparation"."T-30".Raw_Material.ChiliFresh_3.DoseHeld;
      O     "Blend to Preparation"."T-31".Raw_Material.ChiliFresh_3.DoseHeld;
      O     "Blend to Preparation"."T-40".Raw_Material.ChiliFresh_3.DoseHeld;
      O     "Blend to Preparation"."T-41".Raw_Material.ChiliFresh_3.DoseHeld;
      =     "T-08_ChiliFresh_3".IN_Dose_Held;

NETWORK
TITLE = T-08.00 DOSE VALVE CMD
      O(;
      A     "Blend to Preparation"."T-20".Raw_Material.ChiliFresh_3.DoseRun;
      A     "Blend to Preparation"."T-20".Raw_Material.ChiliFresh_3.ValveCMD;
      );
      O(;
      A     "Blend to Preparation"."T-21".Raw_Material.ChiliFresh_3.DoseRun;
      A     "Blend to Preparation"."T-21".Raw_Material.ChiliFresh_3.ValveCMD;
      );
      O(;
      A     "Blend to Preparation"."T-30".Raw_Material.ChiliFresh_3.DoseRun;
      A     "Blend to Preparation"."T-30".Raw_Material.ChiliFresh_3.ValveCMD;
      );
      O(;
      A     "Blend to Preparation"."T-31".Raw_Material.ChiliFresh_3.DoseRun;
      A     "Blend to Preparation"."T-31".Raw_Material.ChiliFresh_3.ValveCMD;
      );
      O(;
      A     "Blend to Preparation"."T-40".Raw_Material.ChiliFresh_3.DoseRun;
      A     "Blend to Preparation"."T-40".Raw_Material.ChiliFresh_3.ValveCMD;
      );
      O(;
      A     "Blend to Preparation"."T-41".Raw_Material.ChiliFresh_3.DoseRun;
      A     "Blend to Preparation"."T-41".Raw_Material.ChiliFresh_3.ValveCMD;
      );
      =     "T-08_ChiliFresh_3".IN_Dose_Valve_Cmd;



NETWORK
TITLE = T-08.00 DOSE Pump CMD
      O(;
      A     "Blend to Preparation"."T-20".Raw_Material.ChiliFresh_3.DoseRun;
      A     "Blend to Preparation"."T-20".Raw_Material.ChiliFresh_3.PumpCMD;
      );
      O(;
      A     "Blend to Preparation"."T-21".Raw_Material.ChiliFresh_3.DoseRun;
      A     "Blend to Preparation"."T-21".Raw_Material.ChiliFresh_3.PumpCMD;
      );
      O(;
      A     "Blend to Preparation"."T-30".Raw_Material.ChiliFresh_3.DoseRun;
      A     "Blend to Preparation"."T-30".Raw_Material.ChiliFresh_3.PumpCMD;
      );
      O(;
      A     "Blend to Preparation"."T-31".Raw_Material.ChiliFresh_3.DoseRun;
      A     "Blend to Preparation"."T-31".Raw_Material.ChiliFresh_3.PumpCMD;
      );
      O(;
      A     "Blend to Preparation"."T-40".Raw_Material.ChiliFresh_3.DoseRun;
      A     "Blend to Preparation"."T-40".Raw_Material.ChiliFresh_3.PumpCMD;
      );
      O(;
      A     "Blend to Preparation"."T-41".Raw_Material.ChiliFresh_3.DoseRun;
      A     "Blend to Preparation"."T-41".Raw_Material.ChiliFresh_3.PumpCMD;
      );
      =     "T-08_ChiliFresh_3".IN_Dose_Pump_Cmd;



NETWORK
TITLE = T-08.00 DOSE PUMP SPEED
// Checking
      O     "Blend to Preparation"."T-20".Raw_Material.ChiliFresh_3.DoseRun;
      JC    SP_08_FROM_20;
      O     "Blend to Preparation"."T-21".Raw_Material.ChiliFresh_3.DoseRun;
      JC    SP_08_FROM_21;
      O     "Blend to Preparation"."T-30".Raw_Material.ChiliFresh_3.DoseRun;
      JC    SP_08_FROM_30;
      O     "Blend to Preparation"."T-31".Raw_Material.ChiliFresh_3.DoseRun;
      JC    SP_08_FROM_31;
      O     "Blend to Preparation"."T-40".Raw_Material.ChiliFresh_3.DoseRun;
      JC    SP_08_FROM_40;
      O     "Blend to Preparation"."T-41".Raw_Material.ChiliFresh_3.DoseRun;
      JC    SP_08_FROM_41;
//Jump to end if Blend not Dosing
      JC    SP_08_SELF;
//Load Set Point
SP_08_FROM_20:L     "Blend to Preparation".Recipe."T-20".ChiliFresh_3.SP_PumpSpeed;
      T     "T-08_ChiliFresh_3".IN_Dose_Pump_Sp;
      JC    SP_08_SELF;
SP_08_FROM_21:L     "Blend to Preparation".Recipe."T-21".ChiliFresh_3.SP_PumpSpeed;
      T     "T-08_ChiliFresh_3".IN_Dose_Pump_Sp;
      JC    SP_08_SELF;
SP_08_FROM_30:L     "Blend to Preparation".Recipe."T-30".ChiliFresh_3.SP_PumpSpeed;
      T     "T-08_ChiliFresh_3".IN_Dose_Pump_Sp;
      JC    SP_08_SELF;
SP_08_FROM_31:L     "Blend to Preparation".Recipe."T-31".ChiliFresh_3.SP_PumpSpeed;
      T     "T-08_ChiliFresh_3".IN_Dose_Pump_Sp;
      JC    SP_08_SELF;
SP_08_FROM_40:L     "Blend to Preparation".Recipe."T-40".ChiliFresh_3.SP_PumpSpeed;
      T     "T-08_ChiliFresh_3".IN_Dose_Pump_Sp;
      JC    SP_08_SELF;
SP_08_FROM_41:L     "Blend to Preparation".Recipe."T-41".ChiliFresh_3.SP_PumpSpeed;
      T     "T-08_ChiliFresh_3".IN_Dose_Pump_Sp;
      JC    SP_08_SELF;
// END
SP_08_SELF:L     "T-08_ChiliFresh_3".IN_Dose_Pump_Sp;
      T     "T-08_ChiliFresh_3".IN_Dose_Pump_Sp;


NETWORK
TITLE = T-08.00 Header Req
// HEADER 1 Req
      O     "Blend to Preparation"."T-20".Raw_Material.ChiliFresh_3.Header1_Req;
      O     "Blend to Preparation"."T-21".Raw_Material.ChiliFresh_3.Header1_Req;
      O     "Blend to Preparation"."T-30".Raw_Material.ChiliFresh_3.Header1_Req;
      O     "Blend to Preparation"."T-31".Raw_Material.ChiliFresh_3.Header1_Req;
      O     "Blend to Preparation"."T-40".Raw_Material.ChiliFresh_3.Header1_Req;
      O     "Blend to Preparation"."T-41".Raw_Material.ChiliFresh_3.Header1_Req;
      =     "T-08_ChiliFresh_3".IN_Dose_Header_1;

// HEADER 2 Req
      O     "Blend to Preparation"."T-20".Raw_Material.ChiliFresh_3.Header2_Req;
      O     "Blend to Preparation"."T-21".Raw_Material.ChiliFresh_3.Header2_Req;
      O     "Blend to Preparation"."T-30".Raw_Material.ChiliFresh_3.Header2_Req;
      O     "Blend to Preparation"."T-31".Raw_Material.ChiliFresh_3.Header2_Req;
      O     "Blend to Preparation"."T-40".Raw_Material.ChiliFresh_3.Header2_Req;
      O     "Blend to Preparation"."T-41".Raw_Material.ChiliFresh_3.Header2_Req;
      =     "T-08_ChiliFresh_3".IN_Dose_Header_2;



REGION Network 101: T-08.00 LineTransferOK
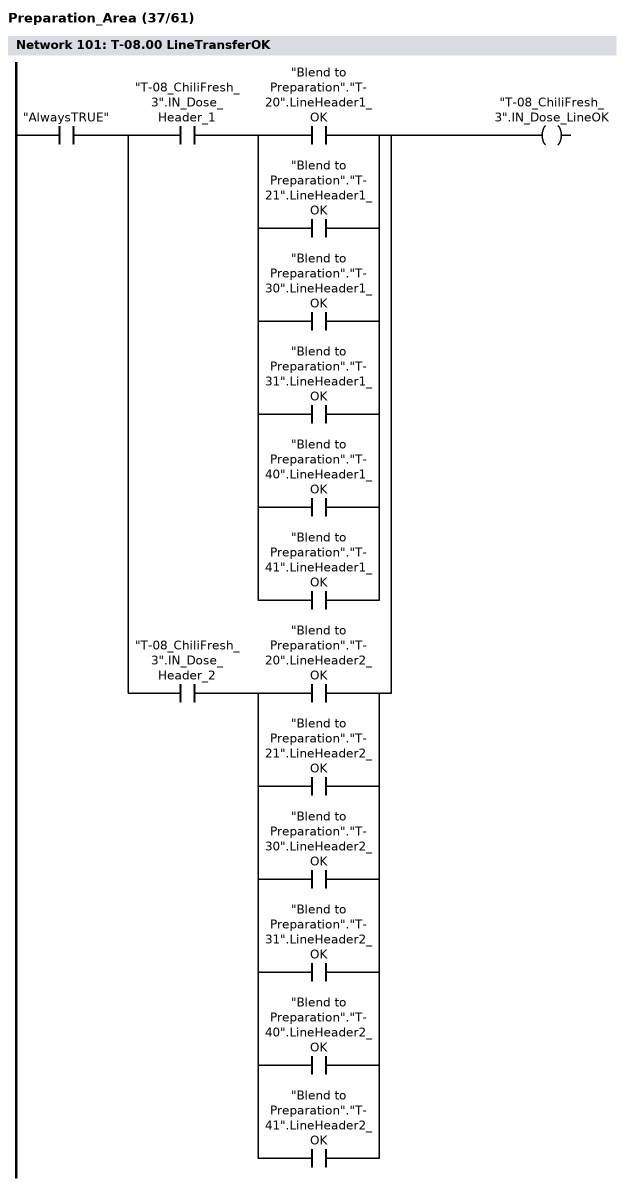
   RUNG wire#powerrail
      Contact( "AlwaysTRUE" )
      wire#w1
      Contact( "T-08_ChiliFresh_3".IN_Dose_Header_1 )
      wire#w2
      Contact( "Blend to Preparation"."T-20".LineHeader1_OK )
      wire#w3
      Coil( "T-08_ChiliFresh_3".IN_Dose_LineOK )
   END_RUNG
   RUNG wire#w2
      Contact( "Blend to Preparation"."T-21".LineHeader1_OK )
   END_RUNG wire#w3
   RUNG wire#w2
      Contact( "Blend to Preparation"."T-30".LineHeader1_OK )
   END_RUNG wire#w3
   RUNG wire#w2
      Contact( "Blend to Preparation"."T-31".LineHeader1_OK )
   END_RUNG wire#w3
   RUNG wire#w2
      Contact( "Blend to Preparation"."T-40".LineHeader1_OK )
   END_RUNG wire#w3
   RUNG wire#w2
      Contact( "Blend to Preparation"."T-41".LineHeader1_OK )
   END_RUNG wire#w3
   RUNG wire#w1
      Contact( "T-08_ChiliFresh_3".IN_Dose_Header_2 )
      wire#w4
      Contact( "Blend to Preparation"."T-20".LineHeader2_OK )
   END_RUNG wire#w3
   RUNG wire#w4
      Contact( "Blend to Preparation"."T-21".LineHeader2_OK )
   END_RUNG wire#w3
   RUNG wire#w4
      Contact( "Blend to Preparation"."T-30".LineHeader2_OK )
   END_RUNG wire#w3
   RUNG wire#w4
      Contact( "Blend to Preparation"."T-31".LineHeader2_OK )
   END_RUNG wire#w3
   RUNG wire#w4
      Contact( "Blend to Preparation"."T-40".LineHeader2_OK )
   END_RUNG wire#w3
   RUNG wire#w4
      Contact( "Blend to Preparation"."T-41".LineHeader2_OK )
   END_RUNG wire#w3
   // the same network as SCL:
   "T-08_ChiliFresh_3".IN_Dose_LineOK := "AlwaysTRUE" AND (("T-08_ChiliFresh_3".IN_Dose_Header_1 AND ("Blend to Preparation"."T-20".LineHeader1_OK OR "Blend to Preparation"."T-21".LineHeader1_OK OR "Blend to Preparation"."T-30".LineHeader1_OK OR "Blend to Preparation"."T-31".LineHeader1_OK OR "Blend to Preparation"."T-40".LineHeader1_OK OR "Blend to Preparation"."T-41".LineHeader1_OK)) OR ("T-08_ChiliFresh_3".IN_Dose_Header_2 AND ("Blend to Preparation"."T-20".LineHeader2_OK OR "Blend to Preparation"."T-21".LineHeader2_OK OR "Blend to Preparation"."T-30".LineHeader2_OK OR "Blend to Preparation"."T-31".LineHeader2_OK OR "Blend to Preparation"."T-40".LineHeader2_OK OR "Blend to Preparation"."T-41".LineHeader2_OK)));
END_REGION

REGION Network 102: T-08____Chili Fresh 3
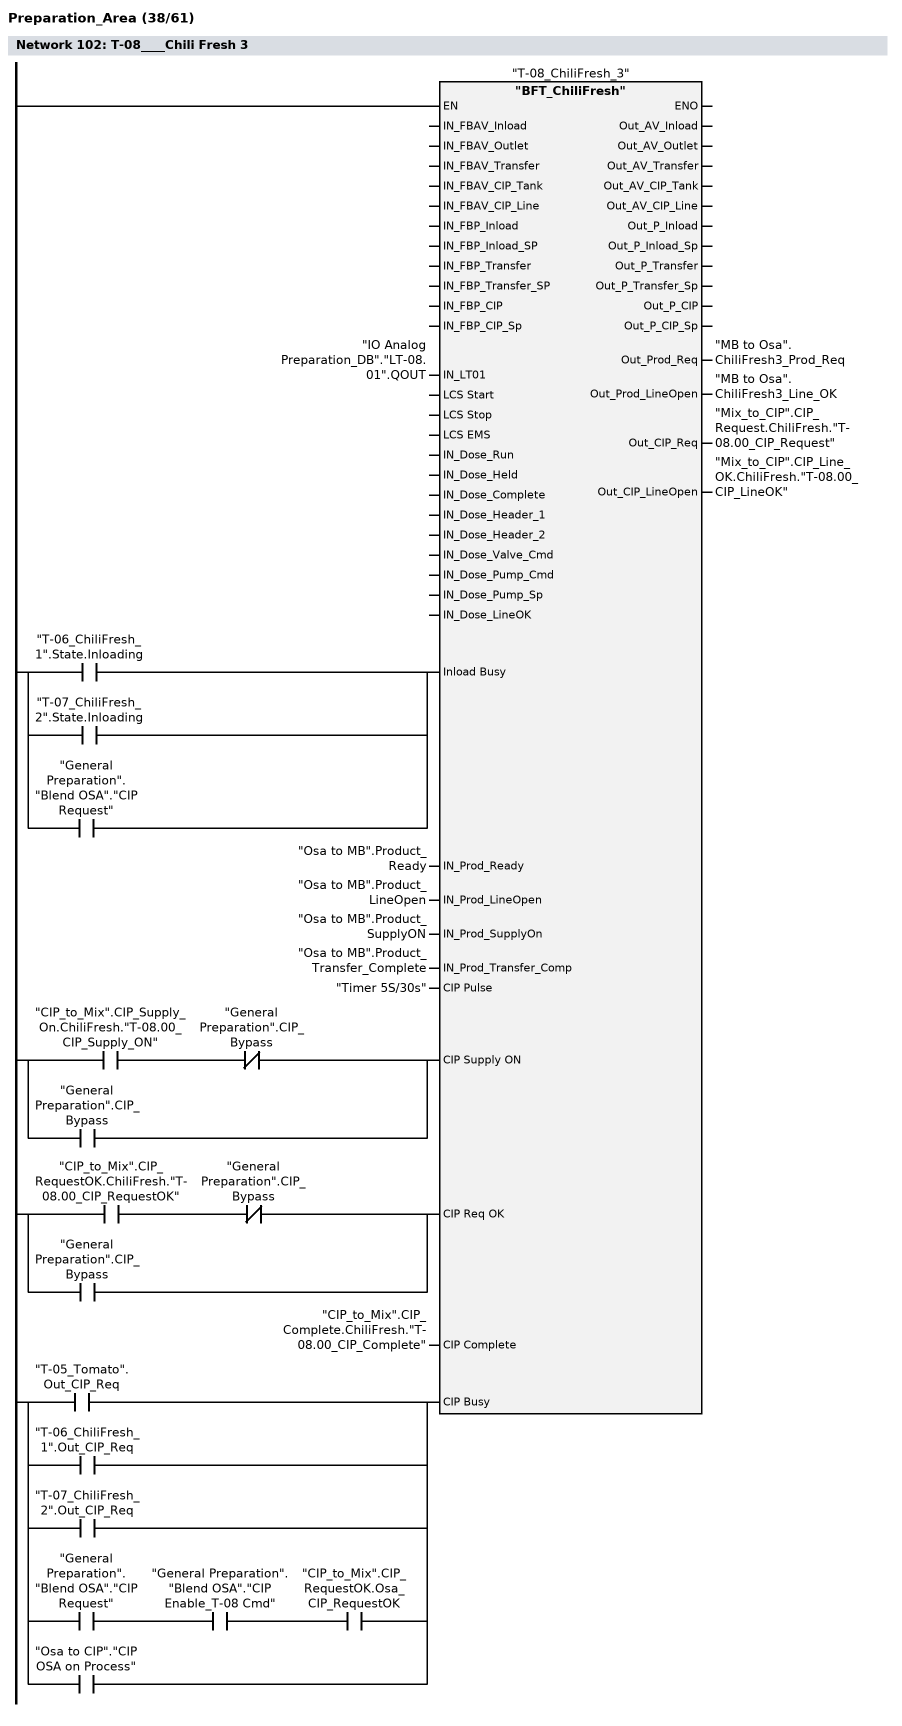
   RUNG wire#powerrail
      "T-08_ChiliFresh_3"("Inload Busy" := wire#w1, "CIP Supply ON" := wire#w2, "CIP Req OK" := wire#w3, "CIP Busy" := wire#w4, IN_FBAV_Inload :=, IN_FBAV_Outlet :=, IN_FBAV_Transfer :=, IN_FBAV_CIP_Tank :=, IN_FBAV_CIP_Line :=, IN_FBP_Inload :=, IN_FBP_Inload_SP :=, IN_FBP_Transfer :=, IN_FBP_Transfer_SP :=, IN_FBP_CIP :=, IN_FBP_CIP_Sp :=, IN_LT01 := "IO Analog Preparation_DB"."LT-08.01".QOUT, "LCS Start" :=, "LCS Stop" :=, "LCS EMS" :=, IN_Dose_Run :=, IN_Dose_Held :=, IN_Dose_Complete :=, IN_Dose_Header_1 :=, IN_Dose_Header_2 :=, IN_Dose_Valve_Cmd :=, IN_Dose_Pump_Cmd :=, IN_Dose_Pump_Sp :=, IN_Dose_LineOK :=, IN_Prod_Ready := "Osa to MB".Product_Ready, IN_Prod_LineOpen := "Osa to MB".Product_LineOpen, IN_Prod_SupplyOn := "Osa to MB".Product_SupplyON, IN_Prod_Transfer_Comp := "Osa to MB".Product_Transfer_Complete, "CIP Pulse" := "Timer 5S/30s", "CIP Complete" := "CIP_to_Mix".CIP_Complete.ChiliFresh."T-08.00_CIP_Complete", Out_AV_Inload =>, Out_AV_Outlet =>, Out_AV_Transfer =>, Out_AV_CIP_Tank =>, Out_AV_CIP_Line =>, Out_P_Inload =>, Out_P_Inload_Sp =>, Out_P_Transfer =>, Out_P_Transfer_Sp =>, Out_P_CIP =>, Out_P_CIP_Sp =>, Out_Prod_Req => "MB to Osa".ChiliFresh3_Prod_Req, Out_Prod_LineOpen => "MB to Osa".ChiliFresh3_Line_OK, Out_CIP_Req => "Mix_to_CIP".CIP_Request.ChiliFresh."T-08.00_CIP_Request", Out_CIP_LineOpen => "Mix_to_CIP".CIP_Line_OK.ChiliFresh."T-08.00_CIP_LineOK")
   END_RUNG
   RUNG wire#powerrail
      Contact( "T-06_ChiliFresh_1".State.Inloading )
   END_RUNG wire#w1
   RUNG wire#powerrail
      Contact( "T-07_ChiliFresh_2".State.Inloading )
   END_RUNG wire#w1
   RUNG wire#powerrail
      Contact( "General Preparation"."Blend OSA"."CIP Request" )
   END_RUNG wire#w1
   RUNG wire#powerrail
      Contact( "CIP_to_Mix".CIP_Supply_On.ChiliFresh."T-08.00_CIP_Supply_ON" )
      I_Contact( "General Preparation".CIP_Bypass )
   END_RUNG wire#w2
   RUNG wire#powerrail
      Contact( "General Preparation".CIP_Bypass )
   END_RUNG wire#w2
   RUNG wire#powerrail
      Contact( "CIP_to_Mix".CIP_RequestOK.ChiliFresh."T-08.00_CIP_RequestOK" )
      I_Contact( "General Preparation".CIP_Bypass )
   END_RUNG wire#w3
   RUNG wire#powerrail
      Contact( "General Preparation".CIP_Bypass )
   END_RUNG wire#w3
   RUNG wire#powerrail
      Contact( "T-05_Tomato".Out_CIP_Req )
   END_RUNG wire#w4
   RUNG wire#powerrail
      Contact( "T-06_ChiliFresh_1".Out_CIP_Req )
   END_RUNG wire#w4
   RUNG wire#powerrail
      Contact( "T-07_ChiliFresh_2".Out_CIP_Req )
   END_RUNG wire#w4
   RUNG wire#powerrail
      Contact( "General Preparation"."Blend OSA"."CIP Request" )
      Contact( "General Preparation"."Blend OSA"."CIP Enable_T-08 Cmd" )
      Contact( "CIP_to_Mix".CIP_RequestOK.Osa_CIP_RequestOK )
   END_RUNG wire#w4
   RUNG wire#powerrail
      Contact( "Osa to CIP"."CIP OSA on Process" )
   END_RUNG wire#w4
   // the same network as SCL:
   "T-08_ChiliFresh_3"(IN_LT01 := "IO Analog Preparation_DB"."LT-08.01".QOUT,   // "BFT_ChiliFresh"
                       "Inload Busy" := "T-06_ChiliFresh_1".State.Inloading OR "T-07_ChiliFresh_2".State.Inloading OR "General Preparation"."Blend OSA"."CIP Request",
                       IN_Prod_Ready := "Osa to MB".Product_Ready,
                       IN_Prod_LineOpen := "Osa to MB".Product_LineOpen,
                       IN_Prod_SupplyOn := "Osa to MB".Product_SupplyON,
                       IN_Prod_Transfer_Comp := "Osa to MB".Product_Transfer_Complete,
                       "CIP Pulse" := "Timer 5S/30s",
                       "CIP Supply ON" := ("CIP_to_Mix".CIP_Supply_On.ChiliFresh."T-08.00_CIP_Supply_ON" AND NOT "General Preparation".CIP_Bypass) OR "General Preparation".CIP_Bypass,
                       "CIP Req OK" := ("CIP_to_Mix".CIP_RequestOK.ChiliFresh."T-08.00_CIP_RequestOK" AND NOT "General Preparation".CIP_Bypass) OR "General Preparation".CIP_Bypass,
                       "CIP Complete" := "CIP_to_Mix".CIP_Complete.ChiliFresh."T-08.00_CIP_Complete",
                       "CIP Busy" := "T-05_Tomato".Out_CIP_Req OR "T-06_ChiliFresh_1".Out_CIP_Req OR "T-07_ChiliFresh_2".Out_CIP_Req OR ("General Preparation"."Blend OSA"."CIP Request" AND "General Preparation"."Blend OSA"."CIP Enable_T-08 Cmd" AND "CIP_to_Mix".CIP_RequestOK.Osa_CIP_RequestOK) OR "Osa to CIP"."CIP OSA on Process",
                       Out_Prod_Req => "MB to Osa".ChiliFresh3_Prod_Req,
                       Out_Prod_LineOpen => "MB to Osa".ChiliFresh3_Line_OK,
                       Out_CIP_Req => "Mix_to_CIP".CIP_Request.ChiliFresh."T-08.00_CIP_Request",
                       Out_CIP_LineOpen => "Mix_to_CIP".CIP_Line_OK.ChiliFresh."T-08.00_CIP_LineOK");
END_REGION

REGION Network 103: T-08.00 Valve Cmd
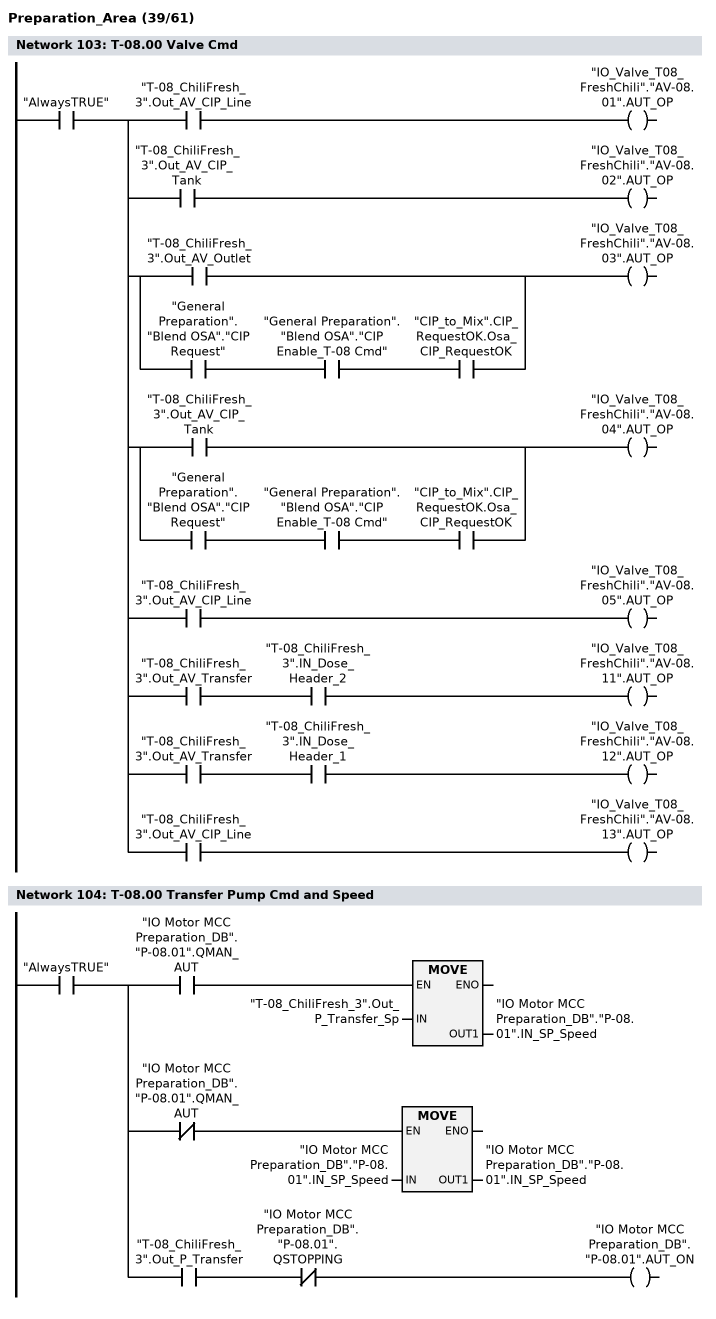
   RUNG wire#powerrail
      Contact( "AlwaysTRUE" )
      wire#w1
      Contact( "T-08_ChiliFresh_3".Out_AV_CIP_Line )
      Coil( "IO_Valve_T08_FreshChili"."AV-08.01".AUT_OP )
   END_RUNG
   RUNG wire#w1
      Contact( "T-08_ChiliFresh_3".Out_AV_CIP_Tank )
      Coil( "IO_Valve_T08_FreshChili"."AV-08.02".AUT_OP )
   END_RUNG
   RUNG wire#w1
      Contact( "T-08_ChiliFresh_3".Out_AV_Outlet )
      wire#w2
      Coil( "IO_Valve_T08_FreshChili"."AV-08.03".AUT_OP )
   END_RUNG
   RUNG wire#w1
      Contact( "General Preparation"."Blend OSA"."CIP Request" )
      Contact( "General Preparation"."Blend OSA"."CIP Enable_T-08 Cmd" )
      Contact( "CIP_to_Mix".CIP_RequestOK.Osa_CIP_RequestOK )
   END_RUNG wire#w2
   RUNG wire#w1
      Contact( "T-08_ChiliFresh_3".Out_AV_CIP_Tank )
      wire#w3
      Coil( "IO_Valve_T08_FreshChili"."AV-08.04".AUT_OP )
   END_RUNG
   RUNG wire#w1
      Contact( "General Preparation"."Blend OSA"."CIP Request" )
      Contact( "General Preparation"."Blend OSA"."CIP Enable_T-08 Cmd" )
      Contact( "CIP_to_Mix".CIP_RequestOK.Osa_CIP_RequestOK )
   END_RUNG wire#w3
   RUNG wire#w1
      Contact( "T-08_ChiliFresh_3".Out_AV_CIP_Line )
      Coil( "IO_Valve_T08_FreshChili"."AV-08.05".AUT_OP )
   END_RUNG
   RUNG wire#w1
      Contact( "T-08_ChiliFresh_3".Out_AV_Transfer )
      Contact( "T-08_ChiliFresh_3".IN_Dose_Header_2 )
      Coil( "IO_Valve_T08_FreshChili"."AV-08.11".AUT_OP )
   END_RUNG
   RUNG wire#w1
      Contact( "T-08_ChiliFresh_3".Out_AV_Transfer )
      Contact( "T-08_ChiliFresh_3".IN_Dose_Header_1 )
      Coil( "IO_Valve_T08_FreshChili"."AV-08.12".AUT_OP )
   END_RUNG
   RUNG wire#w1
      Contact( "T-08_ChiliFresh_3".Out_AV_CIP_Line )
      Coil( "IO_Valve_T08_FreshChili"."AV-08.13".AUT_OP )
   END_RUNG
   // the same network as SCL:
   "IO_Valve_T08_FreshChili"."AV-08.01".AUT_OP := "AlwaysTRUE" AND "T-08_ChiliFresh_3".Out_AV_CIP_Line;
   "IO_Valve_T08_FreshChili"."AV-08.02".AUT_OP := "AlwaysTRUE" AND "T-08_ChiliFresh_3".Out_AV_CIP_Tank;
   "IO_Valve_T08_FreshChili"."AV-08.03".AUT_OP := "AlwaysTRUE" AND ("T-08_ChiliFresh_3".Out_AV_Outlet OR ("General Preparation"."Blend OSA"."CIP Request" AND "General Preparation"."Blend OSA"."CIP Enable_T-08 Cmd" AND "CIP_to_Mix".CIP_RequestOK.Osa_CIP_RequestOK));
   "IO_Valve_T08_FreshChili"."AV-08.04".AUT_OP := "AlwaysTRUE" AND ("T-08_ChiliFresh_3".Out_AV_CIP_Tank OR ("General Preparation"."Blend OSA"."CIP Request" AND "General Preparation"."Blend OSA"."CIP Enable_T-08 Cmd" AND "CIP_to_Mix".CIP_RequestOK.Osa_CIP_RequestOK));
   "IO_Valve_T08_FreshChili"."AV-08.05".AUT_OP := "AlwaysTRUE" AND "T-08_ChiliFresh_3".Out_AV_CIP_Line;
   "IO_Valve_T08_FreshChili"."AV-08.11".AUT_OP := "AlwaysTRUE" AND "T-08_ChiliFresh_3".Out_AV_Transfer AND "T-08_ChiliFresh_3".IN_Dose_Header_2;
   "IO_Valve_T08_FreshChili"."AV-08.12".AUT_OP := "AlwaysTRUE" AND "T-08_ChiliFresh_3".Out_AV_Transfer AND "T-08_ChiliFresh_3".IN_Dose_Header_1;
   "IO_Valve_T08_FreshChili"."AV-08.13".AUT_OP := "AlwaysTRUE" AND "T-08_ChiliFresh_3".Out_AV_CIP_Line;
END_REGION

REGION Network 104: T-08.00 Transfer Pump Cmd and Speed
   RUNG wire#powerrail
      Contact( "AlwaysTRUE" )
      wire#w1
      Contact( "IO Motor MCC Preparation_DB"."P-08.01".QMAN_AUT )
      Move(in := "T-08_ChiliFresh_3".Out_P_Transfer_Sp, out1 => "IO Motor MCC Preparation_DB"."P-08.01".IN_SP_Speed)
   END_RUNG
   RUNG wire#w1
      I_Contact( "IO Motor MCC Preparation_DB"."P-08.01".QMAN_AUT )
      Move(in := "IO Motor MCC Preparation_DB"."P-08.01".IN_SP_Speed, out1 => "IO Motor MCC Preparation_DB"."P-08.01".IN_SP_Speed)
   END_RUNG
   RUNG wire#w1
      Contact( "T-08_ChiliFresh_3".Out_P_Transfer )
      I_Contact( "IO Motor MCC Preparation_DB"."P-08.01".QSTOPPING )
      Coil( "IO Motor MCC Preparation_DB"."P-08.01".AUT_ON )
   END_RUNG
   // the same network as SCL:
   IF "AlwaysTRUE" AND "IO Motor MCC Preparation_DB"."P-08.01".QMAN_AUT THEN
       "IO Motor MCC Preparation_DB"."P-08.01".IN_SP_Speed := "T-08_ChiliFresh_3".Out_P_Transfer_Sp;
   END_IF;
   IF "AlwaysTRUE" AND NOT "IO Motor MCC Preparation_DB"."P-08.01".QMAN_AUT THEN
       "IO Motor MCC Preparation_DB"."P-08.01".IN_SP_Speed := "IO Motor MCC Preparation_DB"."P-08.01".IN_SP_Speed;
   END_IF;
   "IO Motor MCC Preparation_DB"."P-08.01".AUT_ON := "AlwaysTRUE" AND "T-08_ChiliFresh_3".Out_P_Transfer AND NOT "IO Motor MCC Preparation_DB"."P-08.01".QSTOPPING;
END_REGION

REGION Network 105: T-08.00 Feedback Instrument
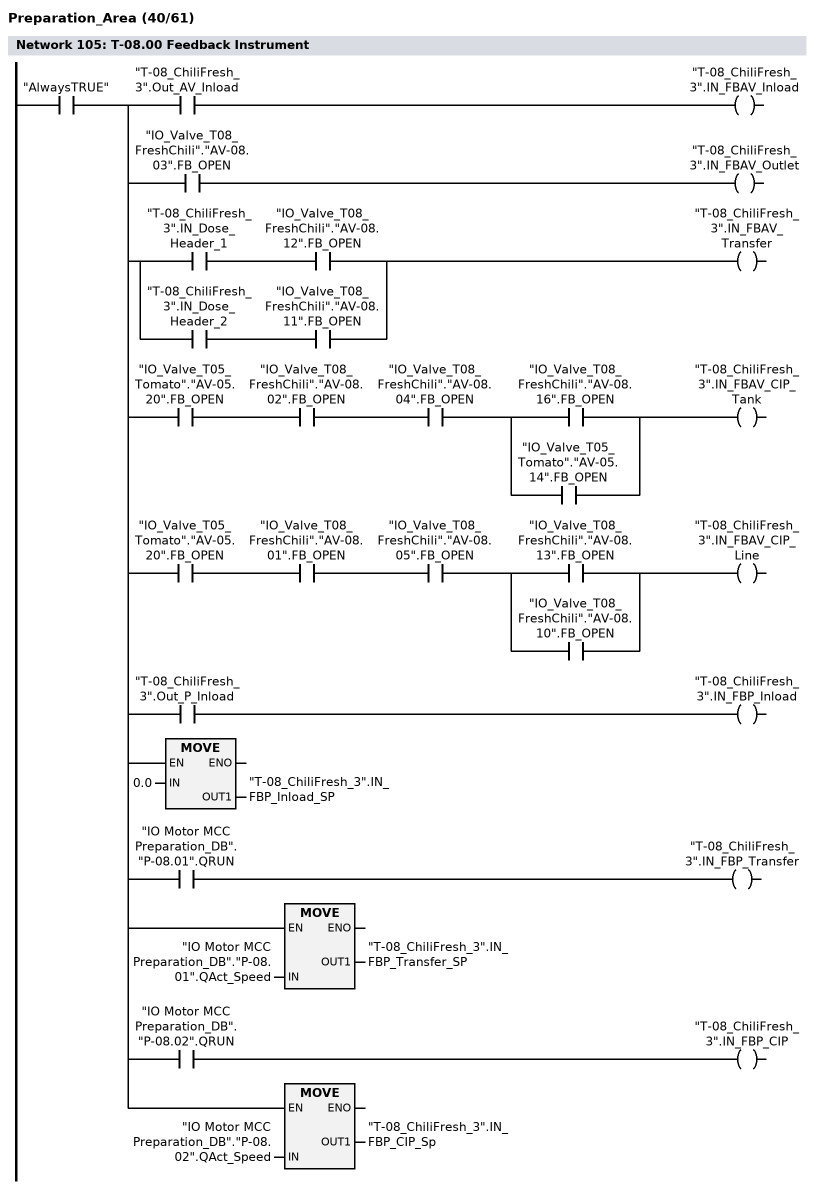
   RUNG wire#powerrail
      Contact( "AlwaysTRUE" )
      wire#w1
      Contact( "T-08_ChiliFresh_3".Out_AV_Inload )
      Coil( "T-08_ChiliFresh_3".IN_FBAV_Inload )
   END_RUNG
   RUNG wire#w1
      Contact( "IO_Valve_T08_FreshChili"."AV-08.03".FB_OPEN )
      Coil( "T-08_ChiliFresh_3".IN_FBAV_Outlet )
   END_RUNG
   RUNG wire#w1
      Contact( "T-08_ChiliFresh_3".IN_Dose_Header_1 )
      Contact( "IO_Valve_T08_FreshChili"."AV-08.12".FB_OPEN )
      wire#w2
      Coil( "T-08_ChiliFresh_3".IN_FBAV_Transfer )
   END_RUNG
   RUNG wire#w1
      Contact( "T-08_ChiliFresh_3".IN_Dose_Header_2 )
      Contact( "IO_Valve_T08_FreshChili"."AV-08.11".FB_OPEN )
   END_RUNG wire#w2
   RUNG wire#w1
      Contact( "IO_Valve_T05_Tomato"."AV-05.20".FB_OPEN )
      Contact( "IO_Valve_T08_FreshChili"."AV-08.02".FB_OPEN )
      Contact( "IO_Valve_T08_FreshChili"."AV-08.04".FB_OPEN )
      wire#w3
      Contact( "IO_Valve_T08_FreshChili"."AV-08.16".FB_OPEN )
      wire#w4
      Coil( "T-08_ChiliFresh_3".IN_FBAV_CIP_Tank )
   END_RUNG
   RUNG wire#w3
      Contact( "IO_Valve_T05_Tomato"."AV-05.14".FB_OPEN )
   END_RUNG wire#w4
   RUNG wire#w1
      Contact( "IO_Valve_T05_Tomato"."AV-05.20".FB_OPEN )
      Contact( "IO_Valve_T08_FreshChili"."AV-08.01".FB_OPEN )
      Contact( "IO_Valve_T08_FreshChili"."AV-08.05".FB_OPEN )
      wire#w5
      Contact( "IO_Valve_T08_FreshChili"."AV-08.13".FB_OPEN )
      wire#w6
      Coil( "T-08_ChiliFresh_3".IN_FBAV_CIP_Line )
   END_RUNG
   RUNG wire#w5
      Contact( "IO_Valve_T08_FreshChili"."AV-08.10".FB_OPEN )
   END_RUNG wire#w6
   RUNG wire#w1
      Contact( "T-08_ChiliFresh_3".Out_P_Inload )
      Coil( "T-08_ChiliFresh_3".IN_FBP_Inload )
   END_RUNG
   RUNG wire#w1
      Move(in := 0.0, out1 => "T-08_ChiliFresh_3".IN_FBP_Inload_SP)
   END_RUNG
   RUNG wire#w1
      Contact( "IO Motor MCC Preparation_DB"."P-08.01".QRUN )
      Coil( "T-08_ChiliFresh_3".IN_FBP_Transfer )
   END_RUNG
   RUNG wire#w1
      Move(in := "IO Motor MCC Preparation_DB"."P-08.01".QAct_Speed, out1 => "T-08_ChiliFresh_3".IN_FBP_Transfer_SP)
   END_RUNG
   RUNG wire#w1
      Contact( "IO Motor MCC Preparation_DB"."P-08.02".QRUN )
      Coil( "T-08_ChiliFresh_3".IN_FBP_CIP )
   END_RUNG
   RUNG wire#w1
      Move(in := "IO Motor MCC Preparation_DB"."P-08.02".QAct_Speed, out1 => "T-08_ChiliFresh_3".IN_FBP_CIP_Sp)
   END_RUNG
   // the same network as SCL:
   "T-08_ChiliFresh_3".IN_FBAV_Inload := "AlwaysTRUE" AND "T-08_ChiliFresh_3".Out_AV_Inload;
   "T-08_ChiliFresh_3".IN_FBAV_Outlet := "AlwaysTRUE" AND "IO_Valve_T08_FreshChili"."AV-08.03".FB_OPEN;
   "T-08_ChiliFresh_3".IN_FBAV_Transfer := "AlwaysTRUE" AND (("T-08_ChiliFresh_3".IN_Dose_Header_1 AND "IO_Valve_T08_FreshChili"."AV-08.12".FB_OPEN) OR ("T-08_ChiliFresh_3".IN_Dose_Header_2 AND "IO_Valve_T08_FreshChili"."AV-08.11".FB_OPEN));
   "T-08_ChiliFresh_3".IN_FBAV_CIP_Tank := "AlwaysTRUE" AND "IO_Valve_T05_Tomato"."AV-05.20".FB_OPEN AND "IO_Valve_T08_FreshChili"."AV-08.02".FB_OPEN AND "IO_Valve_T08_FreshChili"."AV-08.04".FB_OPEN AND ("IO_Valve_T08_FreshChili"."AV-08.16".FB_OPEN OR "IO_Valve_T05_Tomato"."AV-05.14".FB_OPEN);
   "T-08_ChiliFresh_3".IN_FBAV_CIP_Line := "AlwaysTRUE" AND "IO_Valve_T05_Tomato"."AV-05.20".FB_OPEN AND "IO_Valve_T08_FreshChili"."AV-08.01".FB_OPEN AND "IO_Valve_T08_FreshChili"."AV-08.05".FB_OPEN AND ("IO_Valve_T08_FreshChili"."AV-08.13".FB_OPEN OR "IO_Valve_T08_FreshChili"."AV-08.10".FB_OPEN);
   "T-08_ChiliFresh_3".IN_FBP_Inload := "AlwaysTRUE" AND "T-08_ChiliFresh_3".Out_P_Inload;
   IF "AlwaysTRUE" THEN "T-08_ChiliFresh_3".IN_FBP_Inload_SP := 0.0; END_IF;
   "T-08_ChiliFresh_3".IN_FBP_Transfer := "AlwaysTRUE" AND "IO Motor MCC Preparation_DB"."P-08.01".QRUN;
   IF "AlwaysTRUE" THEN
       "T-08_ChiliFresh_3".IN_FBP_Transfer_SP := "IO Motor MCC Preparation_DB"."P-08.01".QAct_Speed;
   END_IF;
   "T-08_ChiliFresh_3".IN_FBP_CIP := "AlwaysTRUE" AND "IO Motor MCC Preparation_DB"."P-08.02".QRUN;
   IF "AlwaysTRUE" THEN
       "T-08_ChiliFresh_3".IN_FBP_CIP_Sp := "IO Motor MCC Preparation_DB"."P-08.02".QAct_Speed;
   END_IF;
END_REGION

REGION Network 106: T-08.00 Comm to Blend
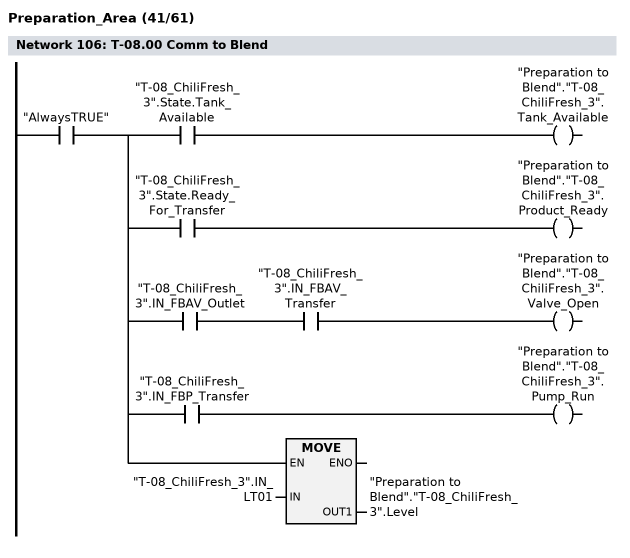
   RUNG wire#powerrail
      Contact( "AlwaysTRUE" )
      wire#w1
      Contact( "T-08_ChiliFresh_3".State.Tank_Available )
      Coil( "Preparation to Blend"."T-08_ChiliFresh_3".Tank_Available )
   END_RUNG
   RUNG wire#w1
      Contact( "T-08_ChiliFresh_3".State.Ready_For_Transfer )
      Coil( "Preparation to Blend"."T-08_ChiliFresh_3".Product_Ready )
   END_RUNG
   RUNG wire#w1
      Contact( "T-08_ChiliFresh_3".IN_FBAV_Outlet )
      Contact( "T-08_ChiliFresh_3".IN_FBAV_Transfer )
      Coil( "Preparation to Blend"."T-08_ChiliFresh_3".Valve_Open )
   END_RUNG
   RUNG wire#w1
      Contact( "T-08_ChiliFresh_3".IN_FBP_Transfer )
      Coil( "Preparation to Blend"."T-08_ChiliFresh_3".Pump_Run )
   END_RUNG
   RUNG wire#w1
      Move(in := "T-08_ChiliFresh_3".IN_LT01, out1 => "Preparation to Blend"."T-08_ChiliFresh_3".Level)
   END_RUNG
   // the same network as SCL:
   "Preparation to Blend"."T-08_ChiliFresh_3".Tank_Available := "AlwaysTRUE" AND "T-08_ChiliFresh_3".State.Tank_Available;
   "Preparation to Blend"."T-08_ChiliFresh_3".Product_Ready := "AlwaysTRUE" AND "T-08_ChiliFresh_3".State.Ready_For_Transfer;
   "Preparation to Blend"."T-08_ChiliFresh_3".Valve_Open := "AlwaysTRUE" AND "T-08_ChiliFresh_3".IN_FBAV_Outlet AND "T-08_ChiliFresh_3".IN_FBAV_Transfer;
   "Preparation to Blend"."T-08_ChiliFresh_3".Pump_Run := "AlwaysTRUE" AND "T-08_ChiliFresh_3".IN_FBP_Transfer;
   IF "AlwaysTRUE" THEN
       "Preparation to Blend"."T-08_ChiliFresh_3".Level := "T-08_ChiliFresh_3".IN_LT01;
   END_IF;
END_REGION

NETWORK
TITLE = T-09.00 DOSE ON OFF
      O     "Blend to Preparation"."T-20".Raw_Material.Garlic.DoseRun;
      O     "Blend to Preparation"."T-21".Raw_Material.Garlic.DoseRun;
      O     "Blend to Preparation"."T-30".Raw_Material.Garlic.DoseRun;
      O     "Blend to Preparation"."T-31".Raw_Material.Garlic.DoseRun;
      O     "Blend to Preparation"."T-40".Raw_Material.Garlic.DoseRun;
      O     "Blend to Preparation"."T-41".Raw_Material.Garlic.DoseRun;
      =     "T-09_Garlic".IN_Dose_Run;

NETWORK
TITLE = T-09.00 DOSE PAUSE
      O     "Blend to Preparation"."T-20".Raw_Material.Garlic.DoseHeld;
      O     "Blend to Preparation"."T-21".Raw_Material.Garlic.DoseHeld;
      O     "Blend to Preparation"."T-30".Raw_Material.Garlic.DoseHeld;
      O     "Blend to Preparation"."T-31".Raw_Material.Garlic.DoseHeld;
      O     "Blend to Preparation"."T-40".Raw_Material.Garlic.DoseHeld;
      O     "Blend to Preparation"."T-41".Raw_Material.Garlic.DoseHeld;
      =     "T-09_Garlic".IN_Dose_Held;

NETWORK
TITLE = T-09.00 DOSE VALVE CMD
      O(;
      A     "Blend to Preparation"."T-20".Raw_Material.Garlic.DoseRun;
      A     "Blend to Preparation"."T-20".Raw_Material.Garlic.ValveCMD;
      );
      O(;
      A     "Blend to Preparation"."T-21".Raw_Material.Garlic.DoseRun;
      A     "Blend to Preparation"."T-21".Raw_Material.Garlic.ValveCMD;
      );
      O(;
      A     "Blend to Preparation"."T-30".Raw_Material.Garlic.DoseRun;
      A     "Blend to Preparation"."T-30".Raw_Material.Garlic.ValveCMD;
      );
      O(;
      A     "Blend to Preparation"."T-31".Raw_Material.Garlic.DoseRun;
      A     "Blend to Preparation"."T-31".Raw_Material.Garlic.ValveCMD;
      );
      O(;
      A     "Blend to Preparation"."T-40".Raw_Material.Garlic.DoseRun;
      A     "Blend to Preparation"."T-40".Raw_Material.Garlic.ValveCMD;
      );
      O(;
      A     "Blend to Preparation"."T-41".Raw_Material.Garlic.DoseRun;
      A     "Blend to Preparation"."T-41".Raw_Material.Garlic.ValveCMD;
      );
      =     "T-09_Garlic".IN_Dose_Valve_Cmd;



NETWORK
TITLE = T-09.00 DOSE Pump CMD
      O(;
      A     "Blend to Preparation"."T-20".Raw_Material.Garlic.DoseRun;
      A     "Blend to Preparation"."T-20".Raw_Material.Garlic.PumpCMD;
      );
      O(;
      A     "Blend to Preparation"."T-21".Raw_Material.Garlic.DoseRun;
      A     "Blend to Preparation"."T-21".Raw_Material.Garlic.PumpCMD;
      );
      O(;
      A     "Blend to Preparation"."T-30".Raw_Material.Garlic.DoseRun;
      A     "Blend to Preparation"."T-30".Raw_Material.Garlic.PumpCMD;
      );
      O(;
      A     "Blend to Preparation"."T-31".Raw_Material.Garlic.DoseRun;
      A     "Blend to Preparation"."T-31".Raw_Material.Garlic.PumpCMD;
      );
      O(;
      A     "Blend to Preparation"."T-40".Raw_Material.Garlic.DoseRun;
      A     "Blend to Preparation"."T-40".Raw_Material.Garlic.PumpCMD;
      );
      O(;
      A     "Blend to Preparation"."T-41".Raw_Material.Garlic.DoseRun;
      A     "Blend to Preparation"."T-41".Raw_Material.Garlic.PumpCMD;
      );
      =     "T-09_Garlic".IN_Dose_Pump_Cmd;



NETWORK
TITLE = T-09.00 DOSE PUMP SPEED
// Checking
      O     "Blend to Preparation"."T-20".Raw_Material.Garlic.DoseRun;
      JC    SP_09_FROM_20;
      O     "Blend to Preparation"."T-21".Raw_Material.Garlic.DoseRun;
      JC    SP_09_FROM_21;
      O     "Blend to Preparation"."T-30".Raw_Material.Garlic.DoseRun;
      JC    SP_09_FROM_30;
      O     "Blend to Preparation"."T-31".Raw_Material.Garlic.DoseRun;
      JC    SP_09_FROM_31;
      O     "Blend to Preparation"."T-40".Raw_Material.Garlic.DoseRun;
      JC    SP_09_FROM_40;
      O     "Blend to Preparation"."T-41".Raw_Material.Garlic.DoseRun;
      JC    SP_09_FROM_41;
//Jump to end if Blend not Dosing
      JC    SP_09_SELF;
//Load Set Point
SP_09_FROM_20:L     "Blend to Preparation".Recipe."T-20".Garlic.SP_PumpSpeed;
      T     "T-09_Garlic".IN_Dose_Pump_Sp;
      JC    SP_09_SELF;
SP_09_FROM_21:L     "Blend to Preparation".Recipe."T-21".Garlic.SP_PumpSpeed;
      T     "T-09_Garlic".IN_Dose_Pump_Sp;
      JC    SP_09_SELF;
SP_09_FROM_30:L     "Blend to Preparation".Recipe."T-30".Garlic.SP_PumpSpeed;
      T     "T-09_Garlic".IN_Dose_Pump_Sp;
      JC    SP_09_SELF;
SP_09_FROM_31:L     "Blend to Preparation".Recipe."T-31".Garlic.SP_PumpSpeed;
      T     "T-09_Garlic".IN_Dose_Pump_Sp;
      JC    SP_09_SELF;
SP_09_FROM_40:L     "Blend to Preparation".Recipe."T-40".Garlic.SP_PumpSpeed;
      T     "T-09_Garlic".IN_Dose_Pump_Sp;
      JC    SP_09_SELF;
SP_09_FROM_41:L     "Blend to Preparation".Recipe."T-41".Garlic.SP_PumpSpeed;
      T     "T-09_Garlic".IN_Dose_Pump_Sp;
      JC    SP_09_SELF;
// END
SP_09_SELF:L     "T-09_Garlic".IN_Dose_Pump_Sp;
      T     "T-09_Garlic".IN_Dose_Pump_Sp;


NETWORK
TITLE = T-09.00 Header Req
// HEADER 1 Req
      O     "Blend to Preparation"."T-20".Raw_Material.Garlic.Header1_Req;
      O     "Blend to Preparation"."T-21".Raw_Material.Garlic.Header1_Req;
      O     "Blend to Preparation"."T-30".Raw_Material.Garlic.Header1_Req;
      O     "Blend to Preparation"."T-31".Raw_Material.Garlic.Header1_Req;
      O     "Blend to Preparation"."T-40".Raw_Material.Garlic.Header1_Req;
      O     "Blend to Preparation"."T-41".Raw_Material.Garlic.Header1_Req;
      =     "T-09_Garlic".IN_Dose_Header_1;

// HEADER 2 Req
      O     "Blend to Preparation"."T-20".Raw_Material.Garlic.Header2_Req;
      O     "Blend to Preparation"."T-21".Raw_Material.Garlic.Header2_Req;
      O     "Blend to Preparation"."T-30".Raw_Material.Garlic.Header2_Req;
      O     "Blend to Preparation"."T-31".Raw_Material.Garlic.Header2_Req;
      O     "Blend to Preparation"."T-40".Raw_Material.Garlic.Header2_Req;
      O     "Blend to Preparation"."T-41".Raw_Material.Garlic.Header2_Req;
      =     "T-09_Garlic".IN_Dose_Header_2;



REGION Network 115: T-09.00 LineTransferOK
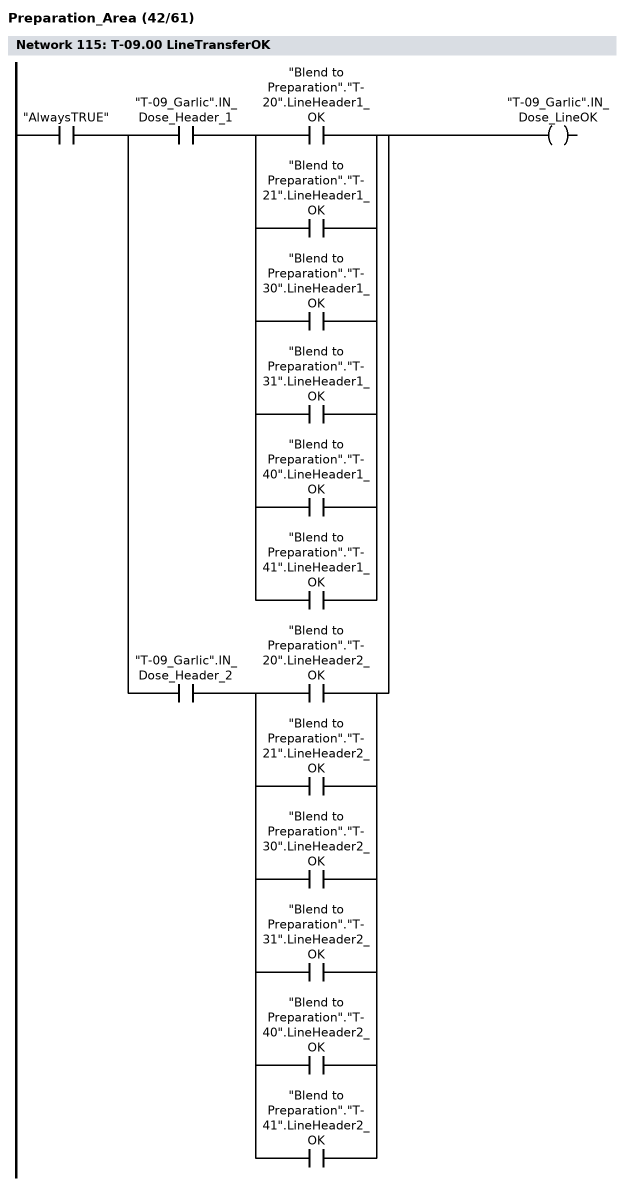
   RUNG wire#powerrail
      Contact( "AlwaysTRUE" )
      wire#w1
      Contact( "T-09_Garlic".IN_Dose_Header_1 )
      wire#w2
      Contact( "Blend to Preparation"."T-20".LineHeader1_OK )
      wire#w3
      Coil( "T-09_Garlic".IN_Dose_LineOK )
   END_RUNG
   RUNG wire#w2
      Contact( "Blend to Preparation"."T-21".LineHeader1_OK )
   END_RUNG wire#w3
   RUNG wire#w2
      Contact( "Blend to Preparation"."T-30".LineHeader1_OK )
   END_RUNG wire#w3
   RUNG wire#w2
      Contact( "Blend to Preparation"."T-31".LineHeader1_OK )
   END_RUNG wire#w3
   RUNG wire#w2
      Contact( "Blend to Preparation"."T-40".LineHeader1_OK )
   END_RUNG wire#w3
   RUNG wire#w2
      Contact( "Blend to Preparation"."T-41".LineHeader1_OK )
   END_RUNG wire#w3
   RUNG wire#w1
      Contact( "T-09_Garlic".IN_Dose_Header_2 )
      wire#w4
      Contact( "Blend to Preparation"."T-20".LineHeader2_OK )
   END_RUNG wire#w3
   RUNG wire#w4
      Contact( "Blend to Preparation"."T-21".LineHeader2_OK )
   END_RUNG wire#w3
   RUNG wire#w4
      Contact( "Blend to Preparation"."T-30".LineHeader2_OK )
   END_RUNG wire#w3
   RUNG wire#w4
      Contact( "Blend to Preparation"."T-31".LineHeader2_OK )
   END_RUNG wire#w3
   RUNG wire#w4
      Contact( "Blend to Preparation"."T-40".LineHeader2_OK )
   END_RUNG wire#w3
   RUNG wire#w4
      Contact( "Blend to Preparation"."T-41".LineHeader2_OK )
   END_RUNG wire#w3
   // the same network as SCL:
   "T-09_Garlic".IN_Dose_LineOK := "AlwaysTRUE" AND (("T-09_Garlic".IN_Dose_Header_1 AND ("Blend to Preparation"."T-20".LineHeader1_OK OR "Blend to Preparation"."T-21".LineHeader1_OK OR "Blend to Preparation"."T-30".LineHeader1_OK OR "Blend to Preparation"."T-31".LineHeader1_OK OR "Blend to Preparation"."T-40".LineHeader1_OK OR "Blend to Preparation"."T-41".LineHeader1_OK)) OR ("T-09_Garlic".IN_Dose_Header_2 AND ("Blend to Preparation"."T-20".LineHeader2_OK OR "Blend to Preparation"."T-21".LineHeader2_OK OR "Blend to Preparation"."T-30".LineHeader2_OK OR "Blend to Preparation"."T-31".LineHeader2_OK OR "Blend to Preparation"."T-40".LineHeader2_OK OR "Blend to Preparation"."T-41".LineHeader2_OK)));
END_REGION

REGION Network 116: T-09.00___Garlic
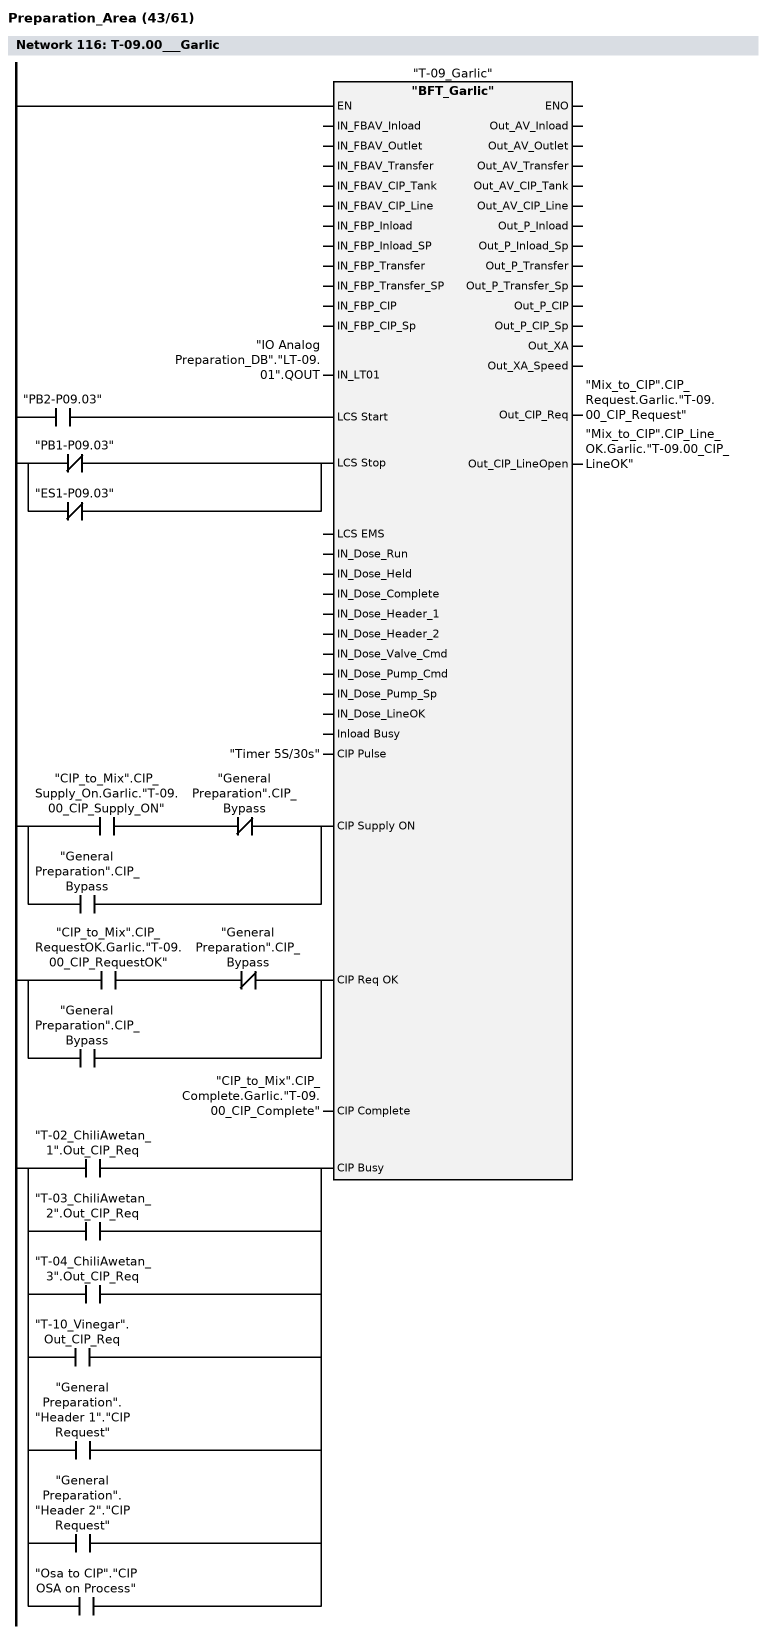
   RUNG wire#powerrail
      "T-09_Garlic"("LCS Start" := wire#w1, "LCS Stop" := wire#w2, "CIP Supply ON" := wire#w3, "CIP Req OK" := wire#w4, "CIP Busy" := wire#w5, IN_FBAV_Inload :=, IN_FBAV_Outlet :=, IN_FBAV_Transfer :=, IN_FBAV_CIP_Tank :=, IN_FBAV_CIP_Line :=, IN_FBP_Inload :=, IN_FBP_Inload_SP :=, IN_FBP_Transfer :=, IN_FBP_Transfer_SP :=, IN_FBP_CIP :=, IN_FBP_CIP_Sp :=, IN_LT01 := "IO Analog Preparation_DB"."LT-09.01".QOUT, "LCS EMS" :=, IN_Dose_Run :=, IN_Dose_Held :=, IN_Dose_Complete :=, IN_Dose_Header_1 :=, IN_Dose_Header_2 :=, IN_Dose_Valve_Cmd :=, IN_Dose_Pump_Cmd :=, IN_Dose_Pump_Sp :=, IN_Dose_LineOK :=, "Inload Busy" :=, "CIP Pulse" := "Timer 5S/30s", "CIP Complete" := "CIP_to_Mix".CIP_Complete.Garlic."T-09.00_CIP_Complete", Out_AV_Inload =>, Out_AV_Outlet =>, Out_AV_Transfer =>, Out_AV_CIP_Tank =>, Out_AV_CIP_Line =>, Out_P_Inload =>, Out_P_Inload_Sp =>, Out_P_Transfer =>, Out_P_Transfer_Sp =>, Out_P_CIP =>, Out_P_CIP_Sp =>, Out_XA =>, Out_XA_Speed =>, Out_CIP_Req => "Mix_to_CIP".CIP_Request.Garlic."T-09.00_CIP_Request", Out_CIP_LineOpen => "Mix_to_CIP".CIP_Line_OK.Garlic."T-09.00_CIP_LineOK")
   END_RUNG
   RUNG wire#powerrail
      Contact( "PB2-P09.03" )
   END_RUNG wire#w1
   RUNG wire#powerrail
      I_Contact( "PB1-P09.03" )
   END_RUNG wire#w2
   RUNG wire#powerrail
      I_Contact( "ES1-P09.03" )
   END_RUNG wire#w2
   RUNG wire#powerrail
      Contact( "CIP_to_Mix".CIP_Supply_On.Garlic."T-09.00_CIP_Supply_ON" )
      I_Contact( "General Preparation".CIP_Bypass )
   END_RUNG wire#w3
   RUNG wire#powerrail
      Contact( "General Preparation".CIP_Bypass )
   END_RUNG wire#w3
   RUNG wire#powerrail
      Contact( "CIP_to_Mix".CIP_RequestOK.Garlic."T-09.00_CIP_RequestOK" )
      I_Contact( "General Preparation".CIP_Bypass )
   END_RUNG wire#w4
   RUNG wire#powerrail
      Contact( "General Preparation".CIP_Bypass )
   END_RUNG wire#w4
   RUNG wire#powerrail
      Contact( "T-02_ChiliAwetan_1".Out_CIP_Req )
   END_RUNG wire#w5
   RUNG wire#powerrail
      Contact( "T-03_ChiliAwetan_2".Out_CIP_Req )
   END_RUNG wire#w5
   RUNG wire#powerrail
      Contact( "T-04_ChiliAwetan_3".Out_CIP_Req )
   END_RUNG wire#w5
   RUNG wire#powerrail
      Contact( "T-10_Vinegar".Out_CIP_Req )
   END_RUNG wire#w5
   RUNG wire#powerrail
      Contact( "General Preparation"."Header 1"."CIP Request" )
   END_RUNG wire#w5
   RUNG wire#powerrail
      Contact( "General Preparation"."Header 2"."CIP Request" )
   END_RUNG wire#w5
   RUNG wire#powerrail
      Contact( "Osa to CIP"."CIP OSA on Process" )
   END_RUNG wire#w5
   // the same network as SCL:
   "T-09_Garlic"(IN_LT01 := "IO Analog Preparation_DB"."LT-09.01".QOUT,   // "BFT_Garlic"
                 "LCS Start" := "PB2-P09.03",
                 "LCS Stop" := NOT "PB1-P09.03" OR NOT "ES1-P09.03",
                 "CIP Pulse" := "Timer 5S/30s",
                 "CIP Supply ON" := ("CIP_to_Mix".CIP_Supply_On.Garlic."T-09.00_CIP_Supply_ON" AND NOT "General Preparation".CIP_Bypass) OR "General Preparation".CIP_Bypass,
                 "CIP Req OK" := ("CIP_to_Mix".CIP_RequestOK.Garlic."T-09.00_CIP_RequestOK" AND NOT "General Preparation".CIP_Bypass) OR "General Preparation".CIP_Bypass,
                 "CIP Complete" := "CIP_to_Mix".CIP_Complete.Garlic."T-09.00_CIP_Complete",
                 "CIP Busy" := "T-02_ChiliAwetan_1".Out_CIP_Req OR "T-03_ChiliAwetan_2".Out_CIP_Req OR "T-04_ChiliAwetan_3".Out_CIP_Req OR "T-10_Vinegar".Out_CIP_Req OR "General Preparation"."Header 1"."CIP Request" OR "General Preparation"."Header 2"."CIP Request" OR "Osa to CIP"."CIP OSA on Process",
                 Out_CIP_Req => "Mix_to_CIP".CIP_Request.Garlic."T-09.00_CIP_Request",
                 Out_CIP_LineOpen => "Mix_to_CIP".CIP_Line_OK.Garlic."T-09.00_CIP_LineOK");
END_REGION

REGION Network 117: T-09.00 Valve Cmd
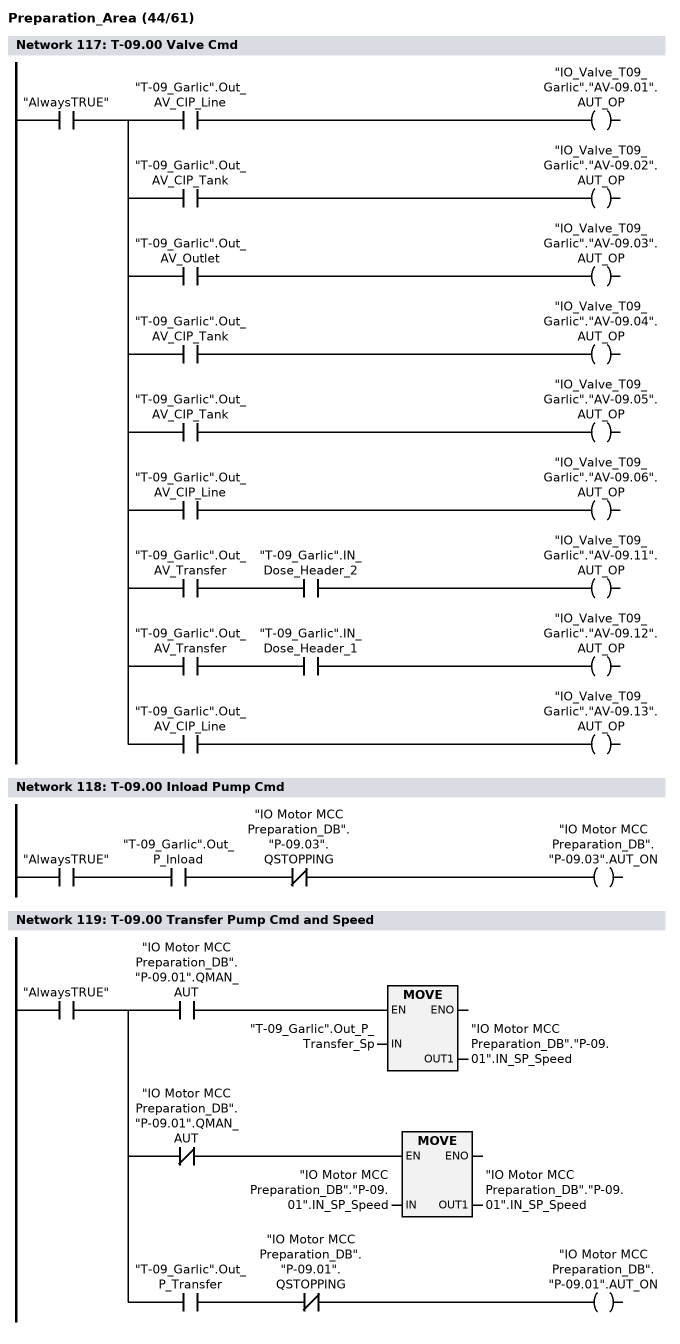
   RUNG wire#powerrail
      Contact( "AlwaysTRUE" )
      wire#w1
      Contact( "T-09_Garlic".Out_AV_CIP_Line )
      Coil( "IO_Valve_T09_Garlic"."AV-09.01".AUT_OP )
   END_RUNG
   RUNG wire#w1
      Contact( "T-09_Garlic".Out_AV_CIP_Tank )
      Coil( "IO_Valve_T09_Garlic"."AV-09.02".AUT_OP )
   END_RUNG
   RUNG wire#w1
      Contact( "T-09_Garlic".Out_AV_Outlet )
      Coil( "IO_Valve_T09_Garlic"."AV-09.03".AUT_OP )
   END_RUNG
   RUNG wire#w1
      Contact( "T-09_Garlic".Out_AV_CIP_Tank )
      Coil( "IO_Valve_T09_Garlic"."AV-09.04".AUT_OP )
   END_RUNG
   RUNG wire#w1
      Contact( "T-09_Garlic".Out_AV_CIP_Tank )
      Coil( "IO_Valve_T09_Garlic"."AV-09.05".AUT_OP )
   END_RUNG
   RUNG wire#w1
      Contact( "T-09_Garlic".Out_AV_CIP_Line )
      Coil( "IO_Valve_T09_Garlic"."AV-09.06".AUT_OP )
   END_RUNG
   RUNG wire#w1
      Contact( "T-09_Garlic".Out_AV_Transfer )
      Contact( "T-09_Garlic".IN_Dose_Header_2 )
      Coil( "IO_Valve_T09_Garlic"."AV-09.11".AUT_OP )
   END_RUNG
   RUNG wire#w1
      Contact( "T-09_Garlic".Out_AV_Transfer )
      Contact( "T-09_Garlic".IN_Dose_Header_1 )
      Coil( "IO_Valve_T09_Garlic"."AV-09.12".AUT_OP )
   END_RUNG
   RUNG wire#w1
      Contact( "T-09_Garlic".Out_AV_CIP_Line )
      Coil( "IO_Valve_T09_Garlic"."AV-09.13".AUT_OP )
   END_RUNG
   // the same network as SCL:
   "IO_Valve_T09_Garlic"."AV-09.01".AUT_OP := "AlwaysTRUE" AND "T-09_Garlic".Out_AV_CIP_Line;
   "IO_Valve_T09_Garlic"."AV-09.02".AUT_OP := "AlwaysTRUE" AND "T-09_Garlic".Out_AV_CIP_Tank;
   "IO_Valve_T09_Garlic"."AV-09.03".AUT_OP := "AlwaysTRUE" AND "T-09_Garlic".Out_AV_Outlet;
   "IO_Valve_T09_Garlic"."AV-09.04".AUT_OP := "AlwaysTRUE" AND "T-09_Garlic".Out_AV_CIP_Tank;
   "IO_Valve_T09_Garlic"."AV-09.05".AUT_OP := "AlwaysTRUE" AND "T-09_Garlic".Out_AV_CIP_Tank;
   "IO_Valve_T09_Garlic"."AV-09.06".AUT_OP := "AlwaysTRUE" AND "T-09_Garlic".Out_AV_CIP_Line;
   "IO_Valve_T09_Garlic"."AV-09.11".AUT_OP := "AlwaysTRUE" AND "T-09_Garlic".Out_AV_Transfer AND "T-09_Garlic".IN_Dose_Header_2;
   "IO_Valve_T09_Garlic"."AV-09.12".AUT_OP := "AlwaysTRUE" AND "T-09_Garlic".Out_AV_Transfer AND "T-09_Garlic".IN_Dose_Header_1;
   "IO_Valve_T09_Garlic"."AV-09.13".AUT_OP := "AlwaysTRUE" AND "T-09_Garlic".Out_AV_CIP_Line;
END_REGION

REGION Network 118: T-09.00 Inload Pump Cmd
   RUNG wire#powerrail
      Contact( "AlwaysTRUE" )
      Contact( "T-09_Garlic".Out_P_Inload )
      I_Contact( "IO Motor MCC Preparation_DB"."P-09.03".QSTOPPING )
      Coil( "IO Motor MCC Preparation_DB"."P-09.03".AUT_ON )
   END_RUNG
   // the same network as SCL:
   "IO Motor MCC Preparation_DB"."P-09.03".AUT_ON := "AlwaysTRUE" AND "T-09_Garlic".Out_P_Inload AND NOT "IO Motor MCC Preparation_DB"."P-09.03".QSTOPPING;
END_REGION

REGION Network 119: T-09.00 Transfer Pump Cmd and Speed
   RUNG wire#powerrail
      Contact( "AlwaysTRUE" )
      wire#w1
      Contact( "IO Motor MCC Preparation_DB"."P-09.01".QMAN_AUT )
      Move(in := "T-09_Garlic".Out_P_Transfer_Sp, out1 => "IO Motor MCC Preparation_DB"."P-09.01".IN_SP_Speed)
   END_RUNG
   RUNG wire#w1
      I_Contact( "IO Motor MCC Preparation_DB"."P-09.01".QMAN_AUT )
      Move(in := "IO Motor MCC Preparation_DB"."P-09.01".IN_SP_Speed, out1 => "IO Motor MCC Preparation_DB"."P-09.01".IN_SP_Speed)
   END_RUNG
   RUNG wire#w1
      Contact( "T-09_Garlic".Out_P_Transfer )
      I_Contact( "IO Motor MCC Preparation_DB"."P-09.01".QSTOPPING )
      Coil( "IO Motor MCC Preparation_DB"."P-09.01".AUT_ON )
   END_RUNG
   // the same network as SCL:
   IF "AlwaysTRUE" AND "IO Motor MCC Preparation_DB"."P-09.01".QMAN_AUT THEN
       "IO Motor MCC Preparation_DB"."P-09.01".IN_SP_Speed := "T-09_Garlic".Out_P_Transfer_Sp;
   END_IF;
   IF "AlwaysTRUE" AND NOT "IO Motor MCC Preparation_DB"."P-09.01".QMAN_AUT THEN
       "IO Motor MCC Preparation_DB"."P-09.01".IN_SP_Speed := "IO Motor MCC Preparation_DB"."P-09.01".IN_SP_Speed;
   END_IF;
   "IO Motor MCC Preparation_DB"."P-09.01".AUT_ON := "AlwaysTRUE" AND "T-09_Garlic".Out_P_Transfer AND NOT "IO Motor MCC Preparation_DB"."P-09.01".QSTOPPING;
END_REGION

REGION Network 120: T-09.00 Agitator Cmd and Speed
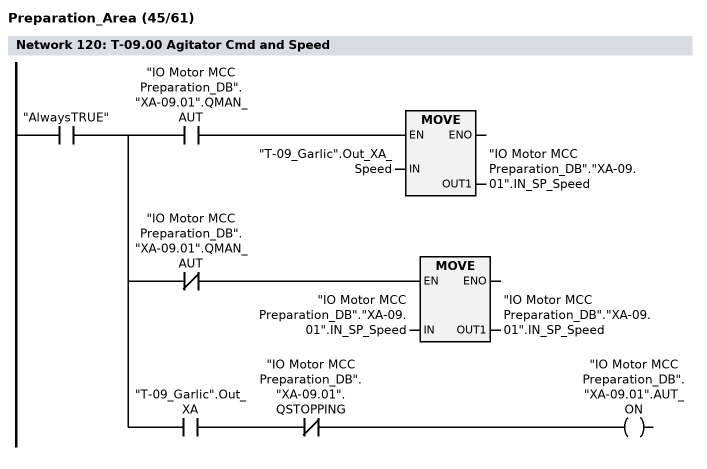
   RUNG wire#powerrail
      Contact( "AlwaysTRUE" )
      wire#w1
      Contact( "IO Motor MCC Preparation_DB"."XA-09.01".QMAN_AUT )
      Move(in := "T-09_Garlic".Out_XA_Speed, out1 => "IO Motor MCC Preparation_DB"."XA-09.01".IN_SP_Speed)
   END_RUNG
   RUNG wire#w1
      I_Contact( "IO Motor MCC Preparation_DB"."XA-09.01".QMAN_AUT )
      Move(in := "IO Motor MCC Preparation_DB"."XA-09.01".IN_SP_Speed, out1 => "IO Motor MCC Preparation_DB"."XA-09.01".IN_SP_Speed)
   END_RUNG
   RUNG wire#w1
      Contact( "T-09_Garlic".Out_XA )
      I_Contact( "IO Motor MCC Preparation_DB"."XA-09.01".QSTOPPING )
      Coil( "IO Motor MCC Preparation_DB"."XA-09.01".AUT_ON )
   END_RUNG
   // the same network as SCL:
   IF "AlwaysTRUE" AND "IO Motor MCC Preparation_DB"."XA-09.01".QMAN_AUT THEN
       "IO Motor MCC Preparation_DB"."XA-09.01".IN_SP_Speed := "T-09_Garlic".Out_XA_Speed;
   END_IF;
   IF "AlwaysTRUE" AND NOT "IO Motor MCC Preparation_DB"."XA-09.01".QMAN_AUT THEN
       "IO Motor MCC Preparation_DB"."XA-09.01".IN_SP_Speed := "IO Motor MCC Preparation_DB"."XA-09.01".IN_SP_Speed;
   END_IF;
   "IO Motor MCC Preparation_DB"."XA-09.01".AUT_ON := "AlwaysTRUE" AND "T-09_Garlic".Out_XA AND NOT "IO Motor MCC Preparation_DB"."XA-09.01".QSTOPPING;
END_REGION

REGION Network 121: T-09.00 Feedback Instrument
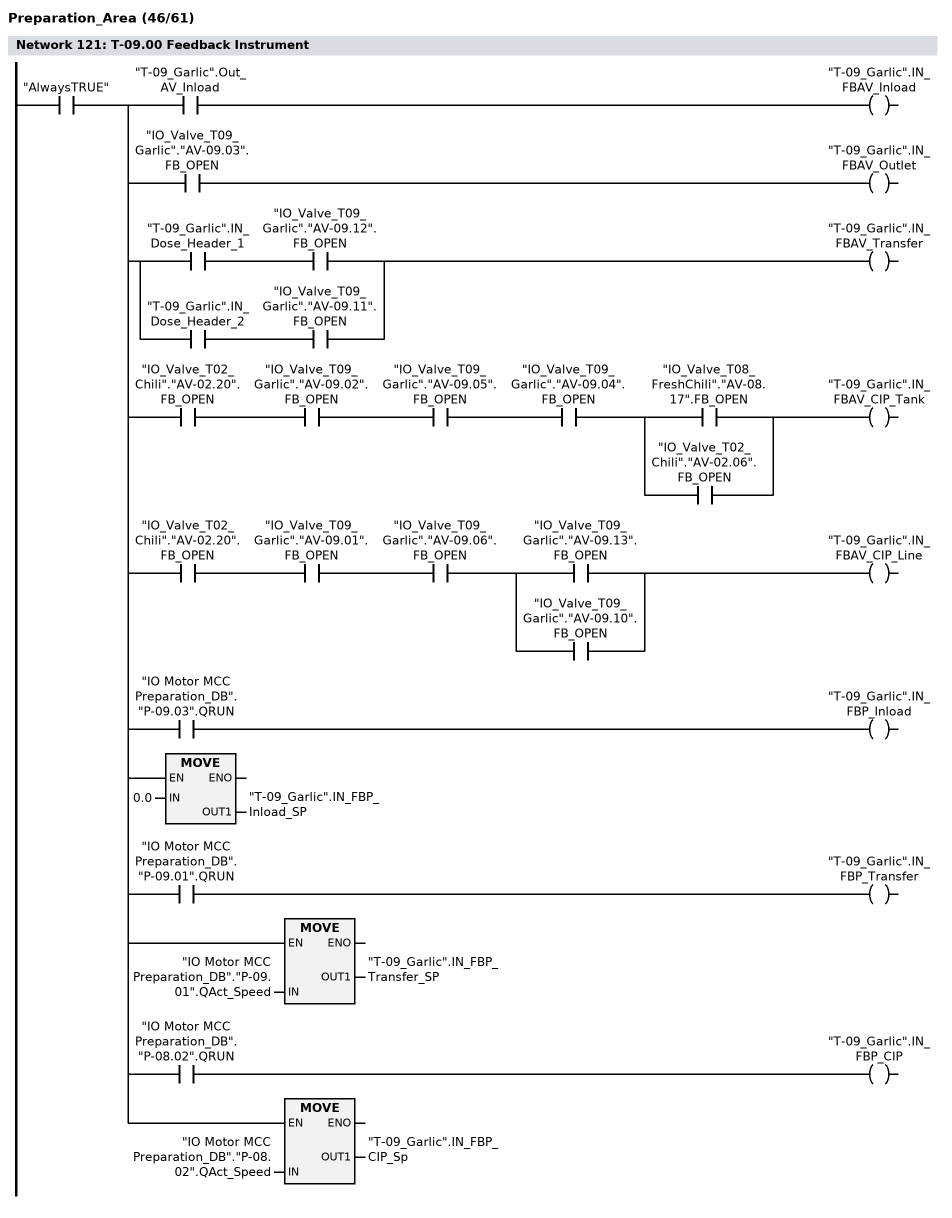
   RUNG wire#powerrail
      Contact( "AlwaysTRUE" )
      wire#w1
      Contact( "T-09_Garlic".Out_AV_Inload )
      Coil( "T-09_Garlic".IN_FBAV_Inload )
   END_RUNG
   RUNG wire#w1
      Contact( "IO_Valve_T09_Garlic"."AV-09.03".FB_OPEN )
      Coil( "T-09_Garlic".IN_FBAV_Outlet )
   END_RUNG
   RUNG wire#w1
      Contact( "T-09_Garlic".IN_Dose_Header_1 )
      Contact( "IO_Valve_T09_Garlic"."AV-09.12".FB_OPEN )
      wire#w2
      Coil( "T-09_Garlic".IN_FBAV_Transfer )
   END_RUNG
   RUNG wire#w1
      Contact( "T-09_Garlic".IN_Dose_Header_2 )
      Contact( "IO_Valve_T09_Garlic"."AV-09.11".FB_OPEN )
   END_RUNG wire#w2
   RUNG wire#w1
      Contact( "IO_Valve_T02_Chili"."AV-02.20".FB_OPEN )
      Contact( "IO_Valve_T09_Garlic"."AV-09.02".FB_OPEN )
      Contact( "IO_Valve_T09_Garlic"."AV-09.05".FB_OPEN )
      Contact( "IO_Valve_T09_Garlic"."AV-09.04".FB_OPEN )
      wire#w3
      Contact( "IO_Valve_T08_FreshChili"."AV-08.17".FB_OPEN )
      wire#w4
      Coil( "T-09_Garlic".IN_FBAV_CIP_Tank )
   END_RUNG
   RUNG wire#w3
      Contact( "IO_Valve_T02_Chili"."AV-02.06".FB_OPEN )
   END_RUNG wire#w4
   RUNG wire#w1
      Contact( "IO_Valve_T02_Chili"."AV-02.20".FB_OPEN )
      Contact( "IO_Valve_T09_Garlic"."AV-09.01".FB_OPEN )
      Contact( "IO_Valve_T09_Garlic"."AV-09.06".FB_OPEN )
      wire#w5
      Contact( "IO_Valve_T09_Garlic"."AV-09.13".FB_OPEN )
      wire#w6
      Coil( "T-09_Garlic".IN_FBAV_CIP_Line )
   END_RUNG
   RUNG wire#w5
      Contact( "IO_Valve_T09_Garlic"."AV-09.10".FB_OPEN )
   END_RUNG wire#w6
   RUNG wire#w1
      Contact( "IO Motor MCC Preparation_DB"."P-09.03".QRUN )
      Coil( "T-09_Garlic".IN_FBP_Inload )
   END_RUNG
   RUNG wire#w1
      Move(in := 0.0, out1 => "T-09_Garlic".IN_FBP_Inload_SP)
   END_RUNG
   RUNG wire#w1
      Contact( "IO Motor MCC Preparation_DB"."P-09.01".QRUN )
      Coil( "T-09_Garlic".IN_FBP_Transfer )
   END_RUNG
   RUNG wire#w1
      Move(in := "IO Motor MCC Preparation_DB"."P-09.01".QAct_Speed, out1 => "T-09_Garlic".IN_FBP_Transfer_SP)
   END_RUNG
   RUNG wire#w1
      Contact( "IO Motor MCC Preparation_DB"."P-08.02".QRUN )
      Coil( "T-09_Garlic".IN_FBP_CIP )
   END_RUNG
   RUNG wire#w1
      Move(in := "IO Motor MCC Preparation_DB"."P-08.02".QAct_Speed, out1 => "T-09_Garlic".IN_FBP_CIP_Sp)
   END_RUNG
   // the same network as SCL:
   "T-09_Garlic".IN_FBAV_Inload := "AlwaysTRUE" AND "T-09_Garlic".Out_AV_Inload;
   "T-09_Garlic".IN_FBAV_Outlet := "AlwaysTRUE" AND "IO_Valve_T09_Garlic"."AV-09.03".FB_OPEN;
   "T-09_Garlic".IN_FBAV_Transfer := "AlwaysTRUE" AND (("T-09_Garlic".IN_Dose_Header_1 AND "IO_Valve_T09_Garlic"."AV-09.12".FB_OPEN) OR ("T-09_Garlic".IN_Dose_Header_2 AND "IO_Valve_T09_Garlic"."AV-09.11".FB_OPEN));
   "T-09_Garlic".IN_FBAV_CIP_Tank := "AlwaysTRUE" AND "IO_Valve_T02_Chili"."AV-02.20".FB_OPEN AND "IO_Valve_T09_Garlic"."AV-09.02".FB_OPEN AND "IO_Valve_T09_Garlic"."AV-09.05".FB_OPEN AND "IO_Valve_T09_Garlic"."AV-09.04".FB_OPEN AND ("IO_Valve_T08_FreshChili"."AV-08.17".FB_OPEN OR "IO_Valve_T02_Chili"."AV-02.06".FB_OPEN);
   "T-09_Garlic".IN_FBAV_CIP_Line := "AlwaysTRUE" AND "IO_Valve_T02_Chili"."AV-02.20".FB_OPEN AND "IO_Valve_T09_Garlic"."AV-09.01".FB_OPEN AND "IO_Valve_T09_Garlic"."AV-09.06".FB_OPEN AND ("IO_Valve_T09_Garlic"."AV-09.13".FB_OPEN OR "IO_Valve_T09_Garlic"."AV-09.10".FB_OPEN);
   "T-09_Garlic".IN_FBP_Inload := "AlwaysTRUE" AND "IO Motor MCC Preparation_DB"."P-09.03".QRUN;
   IF "AlwaysTRUE" THEN "T-09_Garlic".IN_FBP_Inload_SP := 0.0; END_IF;
   "T-09_Garlic".IN_FBP_Transfer := "AlwaysTRUE" AND "IO Motor MCC Preparation_DB"."P-09.01".QRUN;
   IF "AlwaysTRUE" THEN
       "T-09_Garlic".IN_FBP_Transfer_SP := "IO Motor MCC Preparation_DB"."P-09.01".QAct_Speed;
   END_IF;
   "T-09_Garlic".IN_FBP_CIP := "AlwaysTRUE" AND "IO Motor MCC Preparation_DB"."P-08.02".QRUN;
   IF "AlwaysTRUE" THEN
       "T-09_Garlic".IN_FBP_CIP_Sp := "IO Motor MCC Preparation_DB"."P-08.02".QAct_Speed;
   END_IF;
END_REGION

REGION Network 122: T-09.00 Comm to Blend
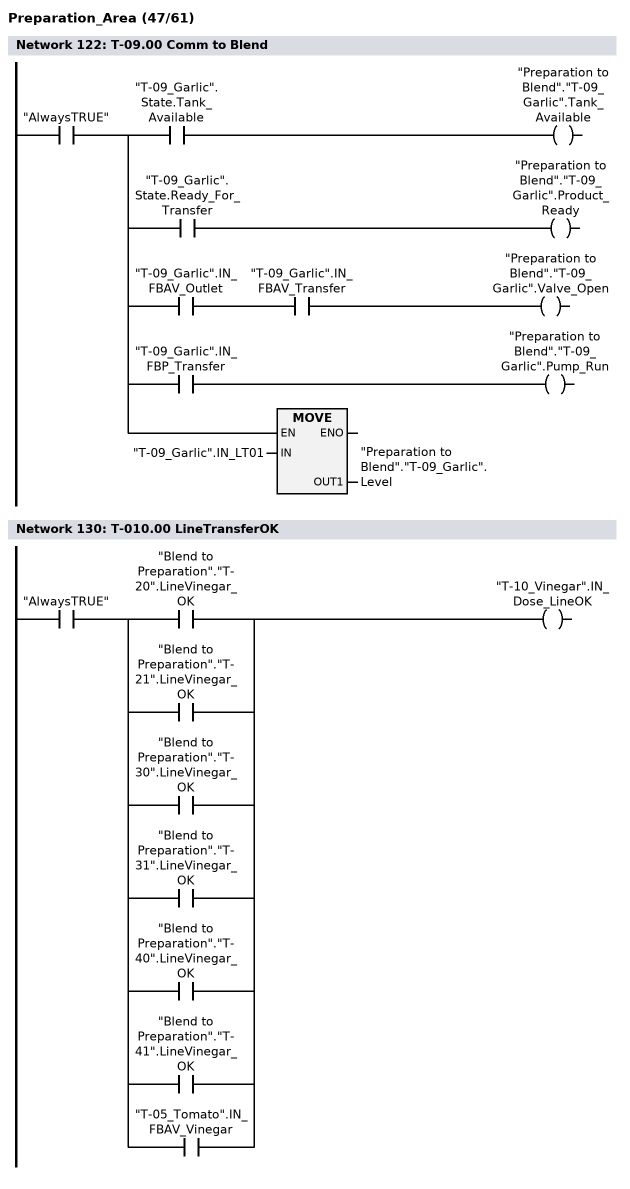
   RUNG wire#powerrail
      Contact( "AlwaysTRUE" )
      wire#w1
      Contact( "T-09_Garlic".State.Tank_Available )
      Coil( "Preparation to Blend"."T-09_Garlic".Tank_Available )
   END_RUNG
   RUNG wire#w1
      Contact( "T-09_Garlic".State.Ready_For_Transfer )
      Coil( "Preparation to Blend"."T-09_Garlic".Product_Ready )
   END_RUNG
   RUNG wire#w1
      Contact( "T-09_Garlic".IN_FBAV_Outlet )
      Contact( "T-09_Garlic".IN_FBAV_Transfer )
      Coil( "Preparation to Blend"."T-09_Garlic".Valve_Open )
   END_RUNG
   RUNG wire#w1
      Contact( "T-09_Garlic".IN_FBP_Transfer )
      Coil( "Preparation to Blend"."T-09_Garlic".Pump_Run )
   END_RUNG
   RUNG wire#w1
      Move(in := "T-09_Garlic".IN_LT01, out1 => "Preparation to Blend"."T-09_Garlic".Level)
   END_RUNG
   // the same network as SCL:
   "Preparation to Blend"."T-09_Garlic".Tank_Available := "AlwaysTRUE" AND "T-09_Garlic".State.Tank_Available;
   "Preparation to Blend"."T-09_Garlic".Product_Ready := "AlwaysTRUE" AND "T-09_Garlic".State.Ready_For_Transfer;
   "Preparation to Blend"."T-09_Garlic".Valve_Open := "AlwaysTRUE" AND "T-09_Garlic".IN_FBAV_Outlet AND "T-09_Garlic".IN_FBAV_Transfer;
   "Preparation to Blend"."T-09_Garlic".Pump_Run := "AlwaysTRUE" AND "T-09_Garlic".IN_FBP_Transfer;
   IF "AlwaysTRUE" THEN "Preparation to Blend"."T-09_Garlic".Level := "T-09_Garlic".IN_LT01; END_IF;
END_REGION

